LIN {X 0,Y 398.014,Z 934.007,A -85,B 0,C 180,E1 13512.725,E2 13512.725} C_VEL
LIN {X 0,Y 394.69,Z 940.929,A -85,B 0,C 180,E1 13512.435,E2 13512.435} C_VEL
LIN {X 0,Y 387.731,Z 954.302,A -85,B 0,C 180,E1 13511.831,E2 13511.831} C_VEL
LIN {X 0,Y 384.258,Z 960.422,A -85,B 0,C 180,E1 13511.522,E2 13511.522} C_VEL
LIN {X 0,Y 377.396,Z 971.989,A -85,B 0,C 180,E1 13510.92,E2 13510.92} C_VEL
LIN {X 0,Y 367.725,Z 986.837,A -85,B 0,C 180,E1 13510.022,E2 13510.022} C_VEL
LIN {X 0,Y 358.47,Z 999.7,A -85,B 0,C 180,E1 13509.091,E2 13509.091} C_VEL
LIN {X 0,Y 349.857,Z 1010.761,A -85,B 0,C 180,E1 13508.133,E2 13508.133} C_VEL
LIN {X 0,Y 342.33,Z 1019.858,A -85,B 0,C 180,E1 13507.215,E2 13507.215} C_VEL
LIN {X 0,Y 335.258,Z 1027.833,A -85,B 0,C 180,E1 13506.25,E2 13506.25} C_VEL
LIN {X 0,Y 328.859,Z 1034.776,A -85,B 0,C 180,E1 13505.234,E2 13505.234} C_VEL
LIN {X 0,Y 322.807,Z 1041.004,A -85,B 0,C 180,E1 13504.122,E2 13504.122} C_VEL
LIN {X 0,Y 317.742,Z 1046.055,A -85,B 0,C 180,E1 13503.067,E2 13503.067} C_VEL
LIN {X 0,Y 313.157,Z 1050.485,A -85,B 0,C 180,E1 13501.963,E2 13501.963} C_VEL
LIN {X 0,Y 312.58,Z 1051.188,A -85,B 0,C 180,E1 13501.741,E2 13501.741} C_VEL
LIN {X 0,Y 311.047,Z 1063.684,A -85,B 0,C 180,E1 13500.267,E2 13500.267} C_VEL
LIN {X 0,Y 309.538,Z 1073.557,A -85,B 0,C 180,E1 13498.797,E2 13498.797} C_VEL
LIN {X 0,Y 307.841,Z 1083.184,A -85,B 0,C 180,E1 13497.021,E2 13497.021} C_VEL
LIN {X 0,Y 306.001,Z 1091.827,A -85,B 0,C 180,E1 13494.938,E2 13494.938} C_VEL
LIN {X 0,Y 304.51,Z 1097.96,A -85,B 0,C 180,E1 13493.022,E2 13493.022} C_VEL
LIN {X 0,Y 303.205,Z 1102.729,A -85,B 0,C 180,E1 13491.084,E2 13491.084} C_VEL
LIN {X 0,Y 302.1,Z 1106.25,A -85,B 0,C 180,E1 13489.125,E2 13489.125} C_VEL
LIN {X 0,Y 301.125,Z 1108.835,A -85,B 0,C 180,E1 13486.95,E2 13486.95} C_VEL
LIN {X 0,Y 300.227,Z 1110.227,A -85,B 0,C 180,E1 13484.151,E2 13484.151} C_VEL
LIN {X 0,Y 299.753,Z 1109.674,A -85,B 0,C 180,E1 13481.726,E2 13481.726} C_VEL
LIN {X 0,Y 299.575,Z 1108.058,A -85,B 0,C 180,E1 13479.689,E2 13479.689} C_VEL
LIN {X 0,Y 299.582,Z 1105.256,A -85,B 0,C 180,E1 13477.6,E2 13477.6} C_VEL
LIN {X 0,Y 299.825,Z 1100.918,A -85,B 0,C 180,E1 13475.363,E2 13475.363} C_VEL
LIN {X 0,Y 300.406,Z 1093.744,A -85,B 0,C 180,E1 13472.714,E2 13472.714} C_VEL
LIN {X 0,Y 300.97,Z 1088.064,A -85,B 0,C 180,E1 13471.032,E2 13471.032} C_VEL
LIN {X 0,Y 302.662,Z 1088.577,A -85,B 0,C 180,E1 13470.076,E2 13470.076} C_VEL
LIN {X 0,Y 308.965,Z 1089.207,A -85,B 0,C 180,E1 13467.505,E2 13467.505} C_VEL
LIN {X 0,Y 318.43,Z 1089.392,A -85,B 0,C 180,E1 13464.485,E2 13464.485} C_VEL
LIN {X 0,Y 330.052,Z 1088.628,A -85,B 0,C 180,E1 13461.689,E2 13461.689} C_VEL
LIN {X 0,Y 343.834,Z 1086.815,A -85,B 0,C 180,E1 13459.132,E2 13459.132} C_VEL
LIN {X 0,Y 345.437,Z 1086.554,A -85,B 0,C 180,E1 13458.874,E2 13458.874} C_VEL
LIN {X 0,Y 335.157,Z 1103.247,A -85,B 0,C 180,E1 13455.24,E2 13455.24} C_VEL
LIN {X 0,Y 325.414,Z 1119.016,A -85,B 0,C 180,E1 13451.115,E2 13451.115} C_VEL
LIN {X 0,Y 317.973,Z 1131.208,A -85,B 0,C 180,E1 13447.29,E2 13447.29} C_VEL
LIN {X 0,Y 310.56,Z 1143.92,A -85,B 0,C 180,E1 13442.483,E2 13442.483} C_VEL
LIN {X 0,Y 305.641,Z 1152.997,A -85,B 0,C 180,E1 13438.32,E2 13438.32} C_VEL
LIN {X 0,Y 301.289,Z 1162.04,A -85,B 0,C 180,E1 13433.263,E2 13433.263} C_VEL
LIN {X 0,Y 298.782,Z 1168.154,A -85,B 0,C 180,E1 13428.944,E2 13428.944} C_VEL
LIN {X 0,Y 297.276,Z 1172.834,A -85,B 0,C 180,E1 13424.813,E2 13424.813} C_VEL
LIN {X 0,Y 296.351,Z 1176.957,A -85,B 0,C 180,E1 13419.865,E2 13419.865} C_VEL
LIN {X 0,Y 296.061,Z 1179.123,A -85,B 0,C 180,E1 13415.623,E2 13415.623} C_VEL
LIN {X 0,Y 295.995,Z 1180.069,A -85,B 0,C 180,E1 13411.938,E2 13411.938} C_VEL
LIN {X 0,Y 295.993,Z 1180.126,A -85,B 0,C 180,E1 13408.454,E2 13408.454} C_VEL
LIN {X 0,Y 296.038,Z 1179.362,A -85,B 0,C 180,E1 13404.964,E2 13404.964} C_VEL
LIN {X 0,Y 296.241,Z 1177.665,A -85,B 0,C 180,E1 13401.266,E2 13401.266} C_VEL
LIN {X 0,Y 296.743,Z 1174.897,A -85,B 0,C 180,E1 13397.351,E2 13397.351} C_VEL
LIN {X 0,Y 298.092,Z 1170.287,A -85,B 0,C 180,E1 13392.633,E2 13392.633} C_VEL
LIN {X 0,Y 300.451,Z 1163.965,A -85,B 0,C 180,E1 13387.913,E2 13387.913} C_VEL
LIN {X 0,Y 303.528,Z 1157.228,A -85,B 0,C 180,E1 13383.808,E2 13383.808} C_VEL
LIN {X 0,Y 308.813,Z 1147.142,A -85,B 0,C 180,E1 13378.801,E2 13378.801} C_VEL
LIN {X 0,Y 314.293,Z 1137.438,A -85,B 0,C 180,E1 13374.845,E2 13374.845} C_VEL
LIN {X 0,Y 321.668,Z 1125.291,A -85,B 0,C 180,E1 13370.649,E2 13370.649} C_VEL
LIN {X 0,Y 329.932,Z 1111.715,A -85,B 0,C 180,E1 13366.775,E2 13366.775} C_VEL
LIN {X 0,Y 339.348,Z 1096.62,A -85,B 0,C 180,E1 13363.125,E2 13363.125} C_VEL
LIN {X 0,Y 349.127,Z 1080.443,A -85,B 0,C 180,E1 13359.87,E2 13359.87} C_VEL
LIN {X 0,Y 359.711,Z 1062.568,A -85,B 0,C 180,E1 13356.821,E2 13356.821} C_VEL
LIN {X 0,Y 369.373,Z 1045.349,A -85,B 0,C 180,E1 13354.352,E2 13354.352} C_VEL
LIN {X 0,Y 372.803,Z 1039.126,A -85,B 0,C 180,E1 13353.53,E2 13353.53} C_VEL
LIN {X 0,Y 375.069,Z 1033.805,A -85,B 0,C 180,E1 13352.741,E2 13352.741} C_VEL
LIN {X 0,Y 378.793,Z 1021.008,A -85,B 0,C 180,E1 13350.448,E2 13350.448} C_VEL
LIN {X 0,Y 381.221,Z 1015.371,A -85,B 0,C 180,E1 13349.727,E2 13349.727} C_VEL
LIN {X 0,Y 391.468,Z 994.143,A -85,B 0,C 180,E1 13347.75,E2 13347.75} C_VEL
LIN {X 0,Y 401.494,Z 971.549,A -85,B 0,C 180,E1 13345.973,E2 13345.973} C_VEL
LIN {X 0,Y 410.028,Z 949.956,A -85,B 0,C 180,E1 13344.557,E2 13344.557} C_VEL
LIN {X 0,Y 418.764,Z 924.964,A -85,B 0,C 180,E1 13343.187,E2 13343.187} C_VEL
LIN {X 0,Y 425.429,Z 902.92,A -85,B 0,C 180,E1 13342.184,E2 13342.184} C_VEL
LIN {X 0,Y 432.132,Z 876.432,A -85,B 0,C 180,E1 13341.205,E2 13341.205} C_VEL
LIN {X 0,Y 440.836,Z 835.745,A -85,B 0,C 180,E1 13340.043,E2 13340.043} C_VEL
LIN {X 0,Y 454.676,Z 767.712,A -85,B 0,C 180,E1 13338.499,E2 13338.499} C_VEL
LIN {X 0,Y 466.705,Z 700.879,A -85,B 0,C 180,E1 13337.159,E2 13337.159} C_VEL
LIN {X 0,Y 476.357,Z 638.132,A -85,B 0,C 180,E1 13336.035,E2 13336.035} C_VEL
LIN {X 0,Y 480.624,Z 605.539,A -85,B 0,C 180,E1 13335.479,E2 13335.479} C_VEL
LIN {X 0,Y 475.05,Z 603.148,A -85,B 0,C 180,E1 13332.397,E2 13332.397} C_VEL
LIN {X 0,Y 471.241,Z 602.431,A -85,B 0,C 180,E1 13329.773,E2 13329.773} C_VEL
LIN {X 0,Y 467.289,Z 604.236,A -85,B 0,C 180,E1 13326.265,E2 13326.265} C_VEL
LIN {X 0,Y 465.287,Z 607.075,A -85,B 0,C 180,E1 13323.696,E2 13323.696} C_VEL
LIN {X 0,Y 463.897,Z 611.957,A -85,B 0,C 180,E1 13320.679,E2 13320.679} C_VEL
LIN {X 0,Y 463.503,Z 617.063,A -85,B 0,C 180,E1 13318.455,E2 13318.455} C_VEL
LIN {X 0,Y 460.723,Z 644.789,A -85,B 0,C 180,E1 13316.36,E2 13316.36} C_VEL
LIN {X 0,Y 457.571,Z 678.937,A -85,B 0,C 180,E1 13313.931,E2 13313.931} C_VEL
LIN {X 0,Y 455.045,Z 708.757,A -85,B 0,C 180,E1 13311.749,E2 13311.749} C_VEL
LIN {X 0,Y 453.418,Z 735.459,A -85,B 0,C 180,E1 13309.502,E2 13309.502} C_VEL
LIN {X 0,Y 452.74,Z 761.032,A -85,B 0,C 180,E1 13307.046,E2 13307.046} C_VEL
LIN {X 0,Y 453.158,Z 782.423,A -85,B 0,C 180,E1 13304.728,E2 13304.728} C_VEL
LIN {X 0,Y 454.662,Z 802.684,A -85,B 0,C 180,E1 13302.3,E2 13302.3} C_VEL
LIN {X 0,Y 455.41,Z 809.682,A -85,B 0,C 180,E1 13301.419,E2 13301.419} C_VEL
LIN {X 0,Y 445.885,Z 851.739,A -85,B 0,C 180,E1 13300.46,E2 13300.46} C_VEL
LIN {X 0,Y 436.683,Z 887.236,A -85,B 0,C 180,E1 13299.465,E2 13299.465} C_VEL
LIN {X 0,Y 426.541,Z 923.447,A -85,B 0,C 180,E1 13298.164,E2 13298.164} C_VEL
LIN {X 0,Y 416.365,Z 957.126,A -85,B 0,C 180,E1 13296.656,E2 13296.656} C_VEL
LIN {X 0,Y 408.565,Z 980.494,A -85,B 0,C 180,E1 13295.386,E2 13295.386} C_VEL
LIN {X 0,Y 400.463,Z 1001.95,A -85,B 0,C 180,E1 13294.003,E2 13294.003} C_VEL
LIN {X 0,Y 390.854,Z 1024.162,A -85,B 0,C 180,E1 13292.264,E2 13292.264} C_VEL
LIN {X 0,Y 380.916,Z 1044.801,A -85,B 0,C 180,E1 13290.321,E2 13290.321} C_VEL
LIN {X 0,Y 370.977,Z 1063.841,A -85,B 0,C 180,E1 13288.196,E2 13288.196} C_VEL
LIN {X 0,Y 360.474,Z 1082.231,A -85,B 0,C 180,E1 13285.73,E2 13285.73} C_VEL
LIN {X 0,Y 349.696,Z 1099.779,A -85,B 0,C 180,E1 13282.911,E2 13282.911} C_VEL
LIN {X 0,Y 339.669,Z 1115.345,A -85,B 0,C 180,E1 13279.935,E2 13279.935} C_VEL
LIN {X 0,Y 329.417,Z 1130.44,A -85,B 0,C 180,E1 13276.447,E2 13276.447} C_VEL
LIN {X 0,Y 320.032,Z 1143.814,A -85,B 0,C 180,E1 13272.682,E2 13272.682} C_VEL
LIN {X 0,Y 311.057,Z 1156.534,A -85,B 0,C 180,E1 13268.34,E2 13268.34} C_VEL
LIN {X 0,Y 303.649,Z 1167.257,A -85,B 0,C 180,E1 13263.811,E2 13263.811} C_VEL
LIN {X 0,Y 297.57,Z 1176.576,A -85,B 0,C 180,E1 13258.935,E2 13258.935} C_VEL
LIN {X 0,Y 293.003,Z 1184.34,A -85,B 0,C 180,E1 13253.743,E2 13253.743} C_VEL
LIN {X 0,Y 290.117,Z 1190.259,A -85,B 0,C 180,E1 13248.596,E2 13248.596} C_VEL
LIN {X 0,Y 288.587,Z 1194.684,A -85,B 0,C 180,E1 13243.42,E2 13243.42} C_VEL
LIN {X 0,Y 288.063,Z 1197.528,A -85,B 0,C 180,E1 13238.581,E2 13238.581} C_VEL
LIN {X 0,Y 287.98,Z 1198.959,A -85,B 0,C 180,E1 13234.179,E2 13234.179} C_VEL
LIN {X 0,Y 287.993,Z 1199.454,A -85,B 0,C 180,E1 13229.799,E2 13229.799} C_VEL
LIN {X 0,Y 287.98,Z 1198.913,A -85,B 0,C 180,E1 13225.617,E2 13225.617} C_VEL
LIN {X 0,Y 288.083,Z 1197.331,A -85,B 0,C 180,E1 13221.012,E2 13221.012} C_VEL
LIN {X 0,Y 288.668,Z 1194.394,A -85,B 0,C 180,E1 13216.17,E2 13216.17} C_VEL
LIN {X 0,Y 290.341,Z 1189.756,A -85,B 0,C 180,E1 13210.901,E2 13210.901} C_VEL
LIN {X 0,Y 293.445,Z 1183.493,A -85,B 0,C 180,E1 13205.649,E2 13205.649} C_VEL
LIN {X 0,Y 298.212,Z 1175.485,A -85,B 0,C 180,E1 13200.468,E2 13200.468} C_VEL
LIN {X 0,Y 304.495,Z 1166.011,A -85,B 0,C 180,E1 13195.609,E2 13195.609} C_VEL
LIN {X 0,Y 312.467,Z 1154.557,A -85,B 0,C 180,E1 13190.918,E2 13190.918} C_VEL
LIN {X 0,Y 321.663,Z 1141.485,A -85,B 0,C 180,E1 13186.606,E2 13186.606} C_VEL
LIN {X 0,Y 331.376,Z 1127.495,A -85,B 0,C 180,E1 13182.84,E2 13182.84} C_VEL
LIN {X 0,Y 342.245,Z 1111.347,A -85,B 0,C 180,E1 13179.264,E2 13179.264} C_VEL
LIN {X 0,Y 353.335,Z 1093.987,A -85,B 0,C 180,E1 13176.104,E2 13176.104} C_VEL
LIN {X 0,Y 364.079,Z 1075.99,A -85,B 0,C 180,E1 13173.393,E2 13173.393} C_VEL
LIN {X 0,Y 375.16,Z 1055.883,A -85,B 0,C 180,E1 13170.882,E2 13170.882} C_VEL
LIN {X 0,Y 385.523,Z 1035.367,A -85,B 0,C 180,E1 13168.759,E2 13168.759} C_VEL
LIN {X 0,Y 395.263,Z 1014.129,A -85,B 0,C 180,E1 13166.925,E2 13166.925} C_VEL
LIN {X 0,Y 404.293,Z 991.925,A -85,B 0,C 180,E1 13165.332,E2 13165.332} C_VEL
LIN {X 0,Y 412.504,Z 968.84,A -85,B 0,C 180,E1 13163.958,E2 13163.958} C_VEL
LIN {X 0,Y 422.561,Z 936.541,A -85,B 0,C 180,E1 13162.394,E2 13162.394} C_VEL
LIN {X 0,Y 432.734,Z 901.343,A -85,B 0,C 180,E1 13161.011,E2 13161.011} C_VEL
LIN {X 0,Y 442.358,Z 865.215,A -85,B 0,C 180,E1 13159.894,E2 13159.894} C_VEL
LIN {X 0,Y 448.761,Z 839.044,A -85,B 0,C 180,E1 13159.229,E2 13159.229} C_VEL
LIN {X 0,Y 440.38,Z 855.925,A -85,B 0,C 180,E1 13158.277,E2 13158.277} C_VEL
LIN {X 0,Y 436.828,Z 863.044,A -85,B 0,C 180,E1 13157.877,E2 13157.877} C_VEL
LIN {X 0,Y 428.321,Z 879.64,A -85,B 0,C 180,E1 13156.903,E2 13156.903} C_VEL
LIN {X 0,Y 424.296,Z 887.378,A -85,B 0,C 180,E1 13156.434,E2 13156.434} C_VEL
LIN {X 0,Y 416.15,Z 902.746,A -85,B 0,C 180,E1 13155.468,E2 13155.468} C_VEL
LIN {X 0,Y 405.614,Z 923.215,A -85,B 0,C 180,E1 13154.348,E2 13154.348} C_VEL
LIN {X 0,Y 398.353,Z 937.989,A -85,B 0,C 180,E1 13153.734,E2 13153.734} C_VEL
LIN {X 0,Y 389.653,Z 954.885,A -85,B 0,C 180,E1 13153.051,E2 13153.051} C_VEL
LIN {X 0,Y 384.55,Z 963.752,A -85,B 0,C 180,E1 13152.616,E2 13152.616} C_VEL
LIN {X 0,Y 377.206,Z 975.718,A -85,B 0,C 180,E1 13151.998,E2 13151.998} C_VEL
LIN {X 0,Y 367.979,Z 989.516,A -85,B 0,C 180,E1 13151.203,E2 13151.203} C_VEL
LIN {X 0,Y 358.299,Z 1002.633,A -85,B 0,C 180,E1 13150.288,E2 13150.288} C_VEL
LIN {X 0,Y 349.026,Z 1014.167,A -85,B 0,C 180,E1 13149.315,E2 13149.315} C_VEL
LIN {X 0,Y 341.264,Z 1023.234,A -85,B 0,C 180,E1 13148.424,E2 13148.424} C_VEL
LIN {X 0,Y 333.496,Z 1031.746,A -85,B 0,C 180,E1 13147.407,E2 13147.407} C_VEL
LIN {X 0,Y 326.372,Z 1039.06,A -85,B 0,C 180,E1 13146.332,E2 13146.332} C_VEL
LIN {X 0,Y 320.329,Z 1045.099,A -85,B 0,C 180,E1 13145.276,E2 13145.276} C_VEL
LIN {X 0,Y 314.812,Z 1050.293,A -85,B 0,C 180,E1 13144.184,E2 13144.184} C_VEL
LIN {X 0,Y 309.371,Z 1055.333,A -85,B 0,C 180,E1 13142.907,E2 13142.907} C_VEL
LIN {X 0,Y 305.378,Z 1058.923,A -85,B 0,C 180,E1 13141.876,E2 13141.876} C_VEL
LIN {X 0,Y 304.821,Z 1059.658,A -85,B 0,C 180,E1 13141.645,E2 13141.645} C_VEL
LIN {X 0,Y 302.974,Z 1071.89,A -85,B 0,C 180,E1 13139.945,E2 13139.945} C_VEL
LIN {X 0,Y 301.247,Z 1081.202,A -85,B 0,C 180,E1 13138.288,E2 13138.288} C_VEL
LIN {X 0,Y 299.578,Z 1089.042,A -85,B 0,C 180,E1 13136.556,E2 13136.556} C_VEL
LIN {X 0,Y 297.743,Z 1096.741,A -85,B 0,C 180,E1 13134.411,E2 13134.411} C_VEL
LIN {X 0,Y 295.893,Z 1103.131,A -85,B 0,C 180,E1 13131.947,E2 13131.947} C_VEL
LIN {X 0,Y 294.592,Z 1107.034,A -85,B 0,C 180,E1 13129.834,E2 13129.834} C_VEL
LIN {X 0,Y 293.583,Z 1109.561,A -85,B 0,C 180,E1 13127.81,E2 13127.81} C_VEL
LIN {X 0,Y 292.779,Z 1110.991,A -85,B 0,C 180,E1 13125.765,E2 13125.765} C_VEL
LIN {X 0,Y 292.193,Z 1111.364,A -85,B 0,C 180,E1 13123.704,E2 13123.704} C_VEL
LIN {X 0,Y 291.808,Z 1110.667,A -85,B 0,C 180,E1 13121.625,E2 13121.625} C_VEL
LIN {X 0,Y 291.624,Z 1108.651,A -85,B 0,C 180,E1 13119.319,E2 13119.319} C_VEL
LIN {X 0,Y 291.718,Z 1104.507,A -85,B 0,C 180,E1 13116.572,E2 13116.572} C_VEL
LIN {X 0,Y 292.073,Z 1099.16,A -85,B 0,C 180,E1 13114.209,E2 13114.209} C_VEL
LIN {X 0,Y 292.669,Z 1092.631,A -85,B 0,C 180,E1 13111.958,E2 13111.958} C_VEL
LIN {X 0,Y 294.265,Z 1093.219,A -85,B 0,C 180,E1 13110.928,E2 13110.928} C_VEL
LIN {X 0,Y 300.147,Z 1094.066,A -85,B 0,C 180,E1 13108.241,E2 13108.241} C_VEL
LIN {X 0,Y 309.579,Z 1094.484,A -85,B 0,C 180,E1 13104.906,E2 13104.906} C_VEL
LIN {X 0,Y 320.998,Z 1093.948,A -85,B 0,C 180,E1 13101.92,E2 13101.92} C_VEL
LIN {X 0,Y 334.828,Z 1092.438,A -85,B 0,C 180,E1 13099.156,E2 13099.156} C_VEL
LIN {X 0,Y 336.547,Z 1092.354,A -85,B 0,C 180,E1 13098.802,E2 13098.802} C_VEL
LIN {X 0,Y 326.253,Z 1108.519,A -85,B 0,C 180,E1 13095.071,E2 13095.071} C_VEL
LIN {X 0,Y 316.861,Z 1122.956,A -85,B 0,C 180,E1 13091.026,E2 13091.026} C_VEL
LIN {X 0,Y 308.275,Z 1136.549,A -85,B 0,C 180,E1 13086.412,E2 13086.412} C_VEL
LIN {X 0,Y 302.07,Z 1146.789,A -85,B 0,C 180,E1 13082.206,E2 13082.206} C_VEL
LIN {X 0,Y 296.312,Z 1157.145,A -85,B 0,C 180,E1 13077.018,E2 13077.018} C_VEL
LIN {X 0,Y 292.881,Z 1164.103,A -85,B 0,C 180,E1 13072.694,E2 13072.694} C_VEL
LIN {X 0,Y 290.325,Z 1170.426,A -85,B 0,C 180,E1 13067.852,E2 13067.852} C_VEL
LIN {X 0,Y 288.843,Z 1175.088,A -85,B 0,C 180,E1 13063.006,E2 13063.006} C_VEL
LIN {X 0,Y 288.275,Z 1177.873,A -85,B 0,C 180,E1 13058.982,E2 13058.982} C_VEL
LIN {X 0,Y 288.051,Z 1179.591,A -85,B 0,C 180,E1 13055.18,E2 13055.18} C_VEL
LIN {X 0,Y 287.997,Z 1180.377,A -85,B 0,C 180,E1 13051.594,E2 13051.594} C_VEL
LIN {X 0,Y 288,Z 1180.344,A -85,B 0,C 180,E1 13048.013,E2 13048.013} C_VEL
LIN {X 0,Y 288.061,Z 1179.491,A -85,B 0,C 180,E1 13044.425,E2 13044.425} C_VEL
LIN {X 0,Y 288.304,Z 1177.709,A -85,B 0,C 180,E1 13040.621,E2 13040.621} C_VEL
LIN {X 0,Y 289.106,Z 1174.226,A -85,B 0,C 180,E1 13035.788,E2 13035.788} C_VEL
LIN {X 0,Y 290.795,Z 1169.062,A -85,B 0,C 180,E1 13030.937,E2 13030.937} C_VEL
LIN {X 0,Y 293.23,Z 1163.369,A -85,B 0,C 180,E1 13026.703,E2 13026.703} C_VEL
LIN {X 0,Y 297.462,Z 1155.059,A -85,B 0,C 180,E1 13021.712,E2 13021.712} C_VEL
LIN {X 0,Y 302.72,Z 1145.684,A -85,B 0,C 180,E1 13017.204,E2 13017.204} C_VEL
LIN {X 0,Y 309.427,Z 1134.853,A -85,B 0,C 180,E1 13012.827,E2 13012.827} C_VEL
LIN {X 0,Y 317.472,Z 1122.037,A -85,B 0,C 180,E1 13008.597,E2 13008.597} C_VEL
LIN {X 0,Y 326.533,Z 1108.194,A -85,B 0,C 180,E1 13004.735,E2 13004.735} C_VEL
LIN {X 0,Y 336.251,Z 1092.902,A -85,B 0,C 180,E1 13001.212,E2 13001.212} C_VEL
LIN {X 0,Y 346.526,Z 1076.682,A -85,B 0,C 180,E1 12998.03,E2 12998.03} C_VEL
LIN {X 0,Y 357.37,Z 1058.563,A -85,B 0,C 180,E1 12995.081,E2 12995.081} C_VEL
LIN {X 0,Y 368.737,Z 1038.738,A -85,B 0,C 180,E1 12992.367,E2 12992.367} C_VEL
LIN {X 0,Y 378.852,Z 1019.807,A -85,B 0,C 180,E1 12990.196,E2 12990.196} C_VEL
LIN {X 0,Y 381.221,Z 1015.371,A -85,B 0,C 180,E1 12989.727,E2 12989.727} C_VEL
LIN {X 0,Y 383.63,Z 1009.691,A -85,B 0,C 180,E1 12989.025,E2 12989.025} C_VEL
LIN {X 0,Y 387.595,Z 995.885,A -85,B 0,C 180,E1 12986.93,E2 12986.93} C_VEL
LIN {X 0,Y 390.035,Z 989.923,A -85,B 0,C 180,E1 12986.29,E2 12986.29} C_VEL
LIN {X 0,Y 399.447,Z 968.502,A -85,B 0,C 180,E1 12984.686,E2 12984.686} C_VEL
LIN {X 0,Y 408.62,Z 945.55,A -85,B 0,C 180,E1 12983.231,E2 12983.231} C_VEL
LIN {X 0,Y 416.974,Z 921.32,A -85,B 0,C 180,E1 12981.968,E2 12981.968} C_VEL
LIN {X 0,Y 424.734,Z 894.931,A -85,B 0,C 180,E1 12980.844,E2 12980.844} C_VEL
LIN {X 0,Y 431.12,Z 868.513,A -85,B 0,C 180,E1 12979.947,E2 12979.947} C_VEL
LIN {X 0,Y 440.685,Z 824.326,A -85,B 0,C 180,E1 12978.776,E2 12978.776} C_VEL
LIN {X 0,Y 454.489,Z 756.835,A -85,B 0,C 180,E1 12977.298,E2 12977.298} C_VEL
LIN {X 0,Y 466.083,Z 692.135,A -85,B 0,C 180,E1 12976.043,E2 12976.043} C_VEL
LIN {X 0,Y 475.398,Z 630.7,A -85,B 0,C 180,E1 12974.973,E2 12974.973} C_VEL
LIN {X 0,Y 477.78,Z 612.645,A -85,B 0,C 180,E1 12974.669,E2 12974.669} C_VEL
LIN {X 0,Y 471.735,Z 610.463,A -85,B 0,C 180,E1 12970.997,E2 12970.997} C_VEL
LIN {X 0,Y 469.775,Z 610.503,A -85,B 0,C 180,E1 12969.556,E2 12969.556} C_VEL
LIN {X 0,Y 466.175,Z 612.244,A -85,B 0,C 180,E1 12966.28,E2 12966.28} C_VEL
LIN {X 0,Y 464.276,Z 614.951,A -85,B 0,C 180,E1 12963.828,E2 12963.828} C_VEL
LIN {X 0,Y 462.901,Z 619.763,A -85,B 0,C 180,E1 12960.866,E2 12960.866} C_VEL
LIN {X 0,Y 462.481,Z 623.861,A -85,B 0,C 180,E1 12959.086,E2 12959.086} C_VEL
LIN {X 0,Y 458.864,Z 656.466,A -85,B 0,C 180,E1 12956.651,E2 12956.651} C_VEL
LIN {X 0,Y 453.696,Z 707.234,A -85,B 0,C 180,E1 12953.014,E2 12953.014} C_VEL
LIN {X 0,Y 451.594,Z 733.311,A -85,B 0,C 180,E1 12950.874,E2 12950.874} C_VEL
LIN {X 0,Y 450.341,Z 757.303,A -85,B 0,C 180,E1 12948.652,E2 12948.652} C_VEL
LIN {X 0,Y 450.094,Z 783.869,A -85,B 0,C 180,E1 12945.839,E2 12945.839} C_VEL
LIN {X 0,Y 451.246,Z 806.631,A -85,B 0,C 180,E1 12943.109,E2 12943.109} C_VEL
LIN {X 0,Y 451.841,Z 813.134,A -85,B 0,C 180,E1 12942.293,E2 12942.293} C_VEL
LIN {X 0,Y 442.11,Z 854.607,A -85,B 0,C 180,E1 12941.348,E2 12941.348} C_VEL
LIN {X 0,Y 432.258,Z 891.855,A -85,B 0,C 180,E1 12940.292,E2 12940.292} C_VEL
LIN {X 0,Y 422.263,Z 926.666,A -85,B 0,C 180,E1 12939.028,E2 12939.028} C_VEL
LIN {X 0,Y 411.783,Z 960.528,A -85,B 0,C 180,E1 12937.501,E2 12937.501} C_VEL
LIN {X 0,Y 403.733,Z 983.613,A -85,B 0,C 180,E1 12936.221,E2 12936.221} C_VEL
LIN {X 0,Y 395.071,Z 1005.133,A -85,B 0,C 180,E1 12934.79,E2 12934.79} C_VEL
LIN {X 0,Y 386.015,Z 1025.532,A -85,B 0,C 180,E1 12933.181,E2 12933.181} C_VEL
LIN {X 0,Y 375.478,Z 1046.604,A -85,B 0,C 180,E1 12931.172,E2 12931.172} C_VEL
LIN {X 0,Y 364.771,Z 1066.143,A -85,B 0,C 180,E1 12928.933,E2 12928.933} C_VEL
LIN {X 0,Y 353.987,Z 1084.438,A -85,B 0,C 180,E1 12926.431,E2 12926.431} C_VEL
LIN {X 0,Y 342.948,Z 1101.76,A -85,B 0,C 180,E1 12923.576,E2 12923.576} C_VEL
LIN {X 0,Y 332.169,Z 1117.662,A -85,B 0,C 180,E1 12920.404,E2 12920.404} C_VEL
LIN {X 0,Y 321.805,Z 1132.381,A -85,B 0,C 180,E1 12916.877,E2 12916.877} C_VEL
LIN {X 0,Y 312.194,Z 1145.64,A -85,B 0,C 180,E1 12913.011,E2 12913.011} C_VEL
LIN {X 0,Y 303.41,Z 1157.484,A -85,B 0,C 180,E1 12908.763,E2 12908.763} C_VEL
LIN {X 0,Y 295.54,Z 1168.424,A -85,B 0,C 180,E1 12903.931,E2 12903.931} C_VEL
LIN {X 0,Y 289.191,Z 1177.765,A -85,B 0,C 180,E1 12898.721,E2 12898.721} C_VEL
LIN {X 0,Y 284.823,Z 1185.039,A -85,B 0,C 180,E1 12893.588,E2 12893.588} C_VEL
LIN {X 0,Y 281.889,Z 1191,A -85,B 0,C 180,E1 12888.079,E2 12888.079} C_VEL
LIN {X 0,Y 280.506,Z 1194.951,A -85,B 0,C 180,E1 12882.975,E2 12882.975} C_VEL
LIN {X 0,Y 280.042,Z 1197.561,A -85,B 0,C 180,E1 12878.002,E2 12878.002} C_VEL
LIN {X 0,Y 279.986,Z 1198.831,A -85,B 0,C 180,E1 12873.683,E2 12873.683} C_VEL
LIN {X 0,Y 279.995,Z 1199.152,A -85,B 0,C 180,E1 12869.25,E2 12869.25} C_VEL
LIN {X 0,Y 279.984,Z 1198.554,A -85,B 0,C 180,E1 12865.081,E2 12865.081} C_VEL
LIN {X 0,Y 280.126,Z 1196.84,A -85,B 0,C 180,E1 12860.34,E2 12860.34} C_VEL
LIN {X 0,Y 280.898,Z 1193.667,A -85,B 0,C 180,E1 12855.147,E2 12855.147} C_VEL
LIN {X 0,Y 282.855,Z 1188.794,A -85,B 0,C 180,E1 12849.729,E2 12849.729} C_VEL
LIN {X 0,Y 286.372,Z 1182.299,A -85,B 0,C 180,E1 12844.342,E2 12844.342} C_VEL
LIN {X 0,Y 291.759,Z 1173.87,A -85,B 0,C 180,E1 12838.957,E2 12838.957} C_VEL
LIN {X 0,Y 298.789,Z 1163.828,A -85,B 0,C 180,E1 12833.913,E2 12833.913} C_VEL
LIN {X 0,Y 307.088,Z 1152.503,A -85,B 0,C 180,E1 12829.346,E2 12829.346} C_VEL
LIN {X 0,Y 316.865,Z 1139.176,A -85,B 0,C 180,E1 12825.019,E2 12825.019} C_VEL
LIN {X 0,Y 327.146,Z 1124.861,A -85,B 0,C 180,E1 12821.245,E2 12821.245} C_VEL
LIN {X 0,Y 338.549,Z 1108.283,A -85,B 0,C 180,E1 12817.669,E2 12817.669} C_VEL
LIN {X 0,Y 350.097,Z 1090.523,A -85,B 0,C 180,E1 12814.527,E2 12814.527} C_VEL
LIN {X 0,Y 361.324,Z 1072.084,A -85,B 0,C 180,E1 12811.834,E2 12811.834} C_VEL
LIN {X 0,Y 372.495,Z 1052.072,A -85,B 0,C 180,E1 12809.421,E2 12809.421} C_VEL
LIN {X 0,Y 383.121,Z 1031.276,A -85,B 0,C 180,E1 12807.344,E2 12807.344} C_VEL
LIN {X 0,Y 393.316,Z 1009.128,A -85,B 0,C 180,E1 12805.511,E2 12805.511} C_VEL
LIN {X 0,Y 402.639,Z 986.298,A -85,B 0,C 180,E1 12803.952,E2 12803.952} C_VEL
LIN {X 0,Y 410.669,Z 963.496,A -85,B 0,C 180,E1 12802.661,E2 12802.661} C_VEL
LIN {X 0,Y 421.216,Z 929.649,A -85,B 0,C 180,E1 12801.105,E2 12801.105} C_VEL
LIN {X 0,Y 431.257,Z 895.039,A -85,B 0,C 180,E1 12799.82,E2 12799.82} C_VEL
LIN {X 0,Y 439.459,Z 864.388,A -85,B 0,C 180,E1 12798.899,E2 12798.899} C_VEL
LIN {X 0,Y 430.817,Z 881.146,A -85,B 0,C 180,E1 12797.98,E2 12797.98} C_VEL
LIN {X 0,Y 425.874,Z 890.299,A -85,B 0,C 180,E1 12797.419,E2 12797.419} C_VEL
LIN {X 0,Y 417.508,Z 905.742,A -85,B 0,C 180,E1 12796.487,E2 12796.487} C_VEL
LIN {X 0,Y 414.318,Z 911.672,A -85,B 0,C 180,E1 12796.153,E2 12796.153} C_VEL
LIN {X 0,Y 406.83,Z 926.023,A -85,B 0,C 180,E1 12795.393,E2 12795.393} C_VEL
LIN {X 0,Y 399.167,Z 941.236,A -85,B 0,C 180,E1 12794.778,E2 12794.778} C_VEL
LIN {X 0,Y 390.874,Z 956.968,A -85,B 0,C 180,E1 12794.18,E2 12794.18} C_VEL
LIN {X 0,Y 385.501,Z 966.155,A -85,B 0,C 180,E1 12793.743,E2 12793.743} C_VEL
LIN {X 0,Y 377.869,Z 978.346,A -85,B 0,C 180,E1 12793.147,E2 12793.147} C_VEL
LIN {X 0,Y 367.971,Z 992.762,A -85,B 0,C 180,E1 12792.342,E2 12792.342} C_VEL
LIN {X 0,Y 357.874,Z 1006.076,A -85,B 0,C 180,E1 12791.442,E2 12791.442} C_VEL
LIN {X 0,Y 348.348,Z 1017.567,A -85,B 0,C 180,E1 12790.502,E2 12790.502} C_VEL
LIN {X 0,Y 340.342,Z 1026.586,A -85,B 0,C 180,E1 12789.64,E2 12789.64} C_VEL
LIN {X 0,Y 332.311,Z 1035.119,A -85,B 0,C 180,E1 12788.653,E2 12788.653} C_VEL
LIN {X 0,Y 324.816,Z 1042.561,A -85,B 0,C 180,E1 12787.588,E2 12787.588} C_VEL
LIN {X 0,Y 317.319,Z 1049.618,A -85,B 0,C 180,E1 12786.332,E2 12786.332} C_VEL
LIN {X 0,Y 311.227,Z 1055.183,A -85,B 0,C 180,E1 12785.144,E2 12785.144} C_VEL
LIN {X 0,Y 305.795,Z 1059.905,A -85,B 0,C 180,E1 12783.937,E2 12783.937} C_VEL
LIN {X 0,Y 301.337,Z 1063.737,A -85,B 0,C 180,E1 12782.812,E2 12782.812} C_VEL
LIN {X 0,Y 298.013,Z 1066.561,A -85,B 0,C 180,E1 12781.923,E2 12781.923} C_VEL
LIN {X 0,Y 296.945,Z 1067.648,A -85,B 0,C 180,E1 12781.495,E2 12781.495} C_VEL
LIN {X 0,Y 295.165,Z 1077.599,A -85,B 0,C 180,E1 12779.903,E2 12779.903} C_VEL
LIN {X 0,Y 293.005,Z 1087.662,A -85,B 0,C 180,E1 12777.849,E2 12777.849} C_VEL
LIN {X 0,Y 291.11,Z 1095.149,A -85,B 0,C 180,E1 12775.864,E2 12775.864} C_VEL
LIN {X 0,Y 289.55,Z 1100.635,A -85,B 0,C 180,E1 12774.024,E2 12774.024} C_VEL
LIN {X 0,Y 288.061,Z 1105.265,A -85,B 0,C 180,E1 12772.019,E2 12772.019} C_VEL
LIN {X 0,Y 286.772,Z 1108.747,A -85,B 0,C 180,E1 12769.96,E2 12769.96} C_VEL
LIN {X 0,Y 285.605,Z 1111.304,A -85,B 0,C 180,E1 12767.632,E2 12767.632} C_VEL
LIN {X 0,Y 284.542,Z 1112.609,A -85,B 0,C 180,E1 12764.719,E2 12764.719} C_VEL
LIN {X 0,Y 283.957,Z 1112.01,A -85,B 0,C 180,E1 12762.16,E2 12762.16} C_VEL
LIN {X 0,Y 283.711,Z 1110.36,A -85,B 0,C 180,E1 12760.01,E2 12760.01} C_VEL
LIN {X 0,Y 283.676,Z 1107.585,A -85,B 0,C 180,E1 12757.843,E2 12757.843} C_VEL
LIN {X 0,Y 283.895,Z 1103.157,A -85,B 0,C 180,E1 12755.443,E2 12755.443} C_VEL
LIN {X 0,Y 284.423,Z 1097.12,A -85,B 0,C 180,E1 12752.955,E2 12752.955} C_VEL
LIN {X 0,Y 286.045,Z 1097.691,A -85,B 0,C 180,E1 12751.842,E2 12751.842} C_VEL
LIN {X 0,Y 293.802,Z 1098.92,A -85,B 0,C 180,E1 12747.933,E2 12747.933} C_VEL
LIN {X 0,Y 304.956,Z 1099.359,A -85,B 0,C 180,E1 12744.062,E2 12744.062} C_VEL
LIN {X 0,Y 317.3,Z 1098.764,A -85,B 0,C 180,E1 12740.931,E2 12740.931} C_VEL
LIN {X 0,Y 327.86,Z 1097.768,A -85,B 0,C 180,E1 12738.795,E2 12738.795} C_VEL
LIN {X 0,Y 317.717,Z 1112.781,A -85,B 0,C 180,E1 12735.083,E2 12735.083} C_VEL
LIN {X 0,Y 308.296,Z 1126.876,A -85,B 0,C 180,E1 12730.914,E2 12730.914} C_VEL
LIN {X 0,Y 299.993,Z 1139.324,A -85,B 0,C 180,E1 12726.392,E2 12726.392} C_VEL
LIN {X 0,Y 293.279,Z 1150.12,A -85,B 0,C 180,E1 12721.673,E2 12721.673} C_VEL
LIN {X 0,Y 288.071,Z 1159.03,A -85,B 0,C 180,E1 12716.825,E2 12716.825} C_VEL
LIN {X 0,Y 284.308,Z 1166.565,A -85,B 0,C 180,E1 12711.802,E2 12711.802} C_VEL
LIN {X 0,Y 281.878,Z 1172.38,A -85,B 0,C 180,E1 12706.7,E2 12706.7} C_VEL
LIN {X 0,Y 280.758,Z 1175.993,A -85,B 0,C 180,E1 12702.55,E2 12702.55} C_VEL
LIN {X 0,Y 280.234,Z 1178.592,A -85,B 0,C 180,E1 12698.414,E2 12698.414} C_VEL
LIN {X 0,Y 280.027,Z 1180.395,A -85,B 0,C 180,E1 12693.688,E2 12693.688} C_VEL
LIN {X 0,Y 279.996,Z 1180.743,A -85,B 0,C 180,E1 12689.184,E2 12689.184} C_VEL
LIN {X 0,Y 280.047,Z 1180.025,A -85,B 0,C 180,E1 12685.087,E2 12685.087} C_VEL
LIN {X 0,Y 280.265,Z 1178.422,A -85,B 0,C 180,E1 12681.178,E2 12681.178} C_VEL
LIN {X 0,Y 280.781,Z 1175.91,A -85,B 0,C 180,E1 12677.247,E2 12677.247} C_VEL
LIN {X 0,Y 281.917,Z 1172.28,A -85,B 0,C 180,E1 12673.095,E2 12673.095} C_VEL
LIN {X 0,Y 284.436,Z 1166.306,A -85,B 0,C 180,E1 12667.908,E2 12667.908} C_VEL
LIN {X 0,Y 288.005,Z 1159.161,A -85,B 0,C 180,E1 12663.158,E2 12663.158} C_VEL
LIN {X 0,Y 292.801,Z 1150.902,A -85,B 0,C 180,E1 12658.62,E2 12658.62} C_VEL
LIN {X 0,Y 299.557,Z 1140.049,A -85,B 0,C 180,E1 12653.789,E2 12653.789} C_VEL
LIN {X 0,Y 306.694,Z 1129.267,A -85,B 0,C 180,E1 12649.799,E2 12649.799} C_VEL
LIN {X 0,Y 316.253,Z 1115.037,A -85,B 0,C 180,E1 12645.425,E2 12645.425} C_VEL
LIN {X 0,Y 325.883,Z 1100.796,A -85,B 0,C 180,E1 12641.795,E2 12641.795} C_VEL
LIN {X 0,Y 336.581,Z 1084.562,A -85,B 0,C 180,E1 12638.351,E2 12638.351} C_VEL
LIN {X 0,Y 346.563,Z 1068.957,A -85,B 0,C 180,E1 12635.554,E2 12635.554} C_VEL
LIN {X 0,Y 357.869,Z 1050.397,A -85,B 0,C 180,E1 12632.759,E2 12632.759} C_VEL
LIN {X 0,Y 367.301,Z 1034.041,A -85,B 0,C 180,E1 12630.662,E2 12630.662} C_VEL
LIN {X 0,Y 379.171,Z 1011.913,A -85,B 0,C 180,E1 12628.27,E2 12628.27} C_VEL
LIN {X 0,Y 388.795,Z 992.43,A -85,B 0,C 180,E1 12626.501,E2 12626.501} C_VEL
LIN {X 0,Y 390.035,Z 989.923,A -85,B 0,C 180,E1 12626.29,E2 12626.29} C_VEL
LIN {X 0,Y 392.491,Z 983.908,A -85,B 0,C 180,E1 12625.667,E2 12625.667} C_VEL
LIN {X 0,Y 396.587,Z 969.193,A -85,B 0,C 180,E1 12623.766,E2 12623.766} C_VEL
LIN {X 0,Y 398.812,Z 962.847,A -85,B 0,C 180,E1 12623.211,E2 12623.211} C_VEL
LIN {X 0,Y 408.102,Z 938.86,A -85,B 0,C 180,E1 12621.791,E2 12621.791} C_VEL
LIN {X 0,Y 416.519,Z 913.858,A -85,B 0,C 180,E1 12620.58,E2 12620.58} C_VEL
LIN {X 0,Y 423.496,Z 889.406,A -85,B 0,C 180,E1 12619.608,E2 12619.608} C_VEL
LIN {X 0,Y 430.89,Z 857.605,A -85,B 0,C 180,E1 12618.617,E2 12618.617} C_VEL
LIN {X 0,Y 442.203,Z 806.427,A -85,B 0,C 180,E1 12617.374,E2 12617.374} C_VEL
LIN {X 0,Y 455.207,Z 742.035,A -85,B 0,C 180,E1 12616.021,E2 12616.021} C_VEL
LIN {X 0,Y 466.31,Z 678.954,A -85,B 0,C 180,E1 12614.846,E2 12614.846} C_VEL
LIN {X 0,Y 474.996,Z 619.88,A -85,B 0,C 180,E1 12613.843,E2 12613.843} C_VEL
LIN {X 0,Y 469.419,Z 618.203,A -85,B 0,C 180,E1 12610.183,E2 12610.183} C_VEL
LIN {X 0,Y 465.161,Z 620.101,A -85,B 0,C 180,E1 12606.418,E2 12606.418} C_VEL
LIN {X 0,Y 463.231,Z 622.821,A -85,B 0,C 180,E1 12603.961,E2 12603.961} C_VEL
LIN {X 0,Y 461.827,Z 627.557,A -85,B 0,C 180,E1 12601.054,E2 12601.054} C_VEL
LIN {X 0,Y 461.448,Z 630.692,A -85,B 0,C 180,E1 12599.721,E2 12599.721} C_VEL
LIN {X 0,Y 457.437,Z 663.325,A -85,B 0,C 180,E1 12597.303,E2 12597.303} C_VEL
LIN {X 0,Y 452.054,Z 710.789,A -85,B 0,C 180,E1 12593.897,E2 12593.897} C_VEL
LIN {X 0,Y 449.564,Z 737.493,A -85,B 0,C 180,E1 12591.702,E2 12591.702} C_VEL
LIN {X 0,Y 447.88,Z 762.647,A -85,B 0,C 180,E1 12589.354,E2 12589.354} C_VEL
LIN {X 0,Y 447.245,Z 789.077,A -85,B 0,C 180,E1 12586.525,E2 12586.525} C_VEL
LIN {X 0,Y 448.069,Z 812.08,A -85,B 0,C 180,E1 12583.736,E2 12583.736} C_VEL
LIN {X 0,Y 448.335,Z 816.53,A -85,B 0,C 180,E1 12583.179,E2 12583.179} C_VEL
LIN {X 0,Y 437.715,Z 860.499,A -85,B 0,C 180,E1 12582.175,E2 12582.175} C_VEL
LIN {X 0,Y 427.717,Z 897.087,A -85,B 0,C 180,E1 12581.112,E2 12581.112} C_VEL
LIN {X 0,Y 417.132,Z 932.794,A -85,B 0,C 180,E1 12579.785,E2 12579.785} C_VEL
LIN {X 0,Y 407.503,Z 962.929,A -85,B 0,C 180,E1 12578.404,E2 12578.404} C_VEL
LIN {X 0,Y 399.61,Z 984.962,A -85,B 0,C 180,E1 12577.18,E2 12577.18} C_VEL
LIN {X 0,Y 390.494,Z 1006.844,A -85,B 0,C 180,E1 12575.716,E2 12575.716} C_VEL
LIN {X 0,Y 380.275,Z 1028.649,A -85,B 0,C 180,E1 12573.953,E2 12573.953} C_VEL
LIN {X 0,Y 370.124,Z 1048.398,A -85,B 0,C 180,E1 12572.048,E2 12572.048} C_VEL
LIN {X 0,Y 359.175,Z 1067.631,A -85,B 0,C 180,E1 12569.807,E2 12569.807} C_VEL
LIN {X 0,Y 347.816,Z 1086.064,A -85,B 0,C 180,E1 12567.227,E2 12567.227} C_VEL
LIN {X 0,Y 336.78,Z 1102.879,A -85,B 0,C 180,E1 12564.414,E2 12564.414} C_VEL
LIN {X 0,Y 325.756,Z 1118.583,A -85,B 0,C 180,E1 12561.223,E2 12561.223} C_VEL
LIN {X 0,Y 315.127,Z 1133.003,A -85,B 0,C 180,E1 12557.668,E2 12557.668} C_VEL
LIN {X 0,Y 305.621,Z 1145.679,A -85,B 0,C 180,E1 12553.911,E2 12553.911} C_VEL
LIN {X 0,Y 296.142,Z 1158.014,A -85,B 0,C 180,E1 12549.398,E2 12549.398} C_VEL
LIN {X 0,Y 288.301,Z 1168.379,A -85,B 0,C 180,E1 12544.662,E2 12544.662} C_VEL
LIN {X 0,Y 281.659,Z 1177.717,A -85,B 0,C 180,E1 12539.331,E2 12539.331} C_VEL
LIN {X 0,Y 276.927,Z 1185.174,A -85,B 0,C 180,E1 12533.85,E2 12533.85} C_VEL
LIN {X 0,Y 273.987,Z 1190.857,A -85,B 0,C 180,E1 12528.405,E2 12528.405} C_VEL
LIN {X 0,Y 272.529,Z 1194.809,A -85,B 0,C 180,E1 12523.146,E2 12523.146} C_VEL
LIN {X 0,Y 272.045,Z 1197.363,A -85,B 0,C 180,E1 12518.026,E2 12518.026} C_VEL
LIN {X 0,Y 271.991,Z 1198.66,A -85,B 0,C 180,E1 12513.369,E2 12513.369} C_VEL
LIN {X 0,Y 272.003,Z 1198.87,A -85,B 0,C 180,E1 12508.944,E2 12508.944} C_VEL
LIN {X 0,Y 271.991,Z 1198.192,A -85,B 0,C 180,E1 12504.513,E2 12504.513} C_VEL
LIN {X 0,Y 272.181,Z 1196.345,A -85,B 0,C 180,E1 12499.627,E2 12499.627} C_VEL
LIN {X 0,Y 273.111,Z 1193.053,A -85,B 0,C 180,E1 12494.278,E2 12494.278} C_VEL
LIN {X 0,Y 275.344,Z 1188.045,A -85,B 0,C 180,E1 12488.704,E2 12488.704} C_VEL
LIN {X 0,Y 279.241,Z 1181.365,A -85,B 0,C 180,E1 12483.179,E2 12483.179} C_VEL
LIN {X 0,Y 285.086,Z 1172.786,A -85,B 0,C 180,E1 12477.701,E2 12477.701} C_VEL
LIN {X 0,Y 292.689,Z 1162.518,A -85,B 0,C 180,E1 12472.546,E2 12472.546} C_VEL
LIN {X 0,Y 301.468,Z 1150.989,A -85,B 0,C 180,E1 12467.932,E2 12467.932} C_VEL
LIN {X 0,Y 311.391,Z 1138.026,A -85,B 0,C 180,E1 12463.738,E2 12463.738} C_VEL
LIN {X 0,Y 322.12,Z 1123.542,A -85,B 0,C 180,E1 12459.938,E2 12459.938} C_VEL
LIN {X 0,Y 333.413,Z 1107.635,A -85,B 0,C 180,E1 12456.511,E2 12456.511} C_VEL
LIN {X 0,Y 345.291,Z 1089.938,A -85,B 0,C 180,E1 12453.381,E2 12453.381} C_VEL
LIN {X 0,Y 357.103,Z 1071.044,A -85,B 0,C 180,E1 12450.637,E2 12450.637} C_VEL
LIN {X 0,Y 368.765,Z 1050.659,A -85,B 0,C 180,E1 12448.207,E2 12448.207} C_VEL
LIN {X 0,Y 379.785,Z 1029.506,A -85,B 0,C 180,E1 12446.13,E2 12446.13} C_VEL
LIN {X 0,Y 390.097,Z 1007.486,A -85,B 0,C 180,E1 12444.342,E2 12444.342} C_VEL
LIN {X 0,Y 399.508,Z 984.901,A -85,B 0,C 180,E1 12442.826,E2 12442.826} C_VEL
LIN {X 0,Y 407.923,Z 961.478,A -85,B 0,C 180,E1 12441.528,E2 12441.528} C_VEL
LIN {X 0,Y 418.532,Z 927.897,A -85,B 0,C 180,E1 12440.022,E2 12440.022} C_VEL
LIN {X 0,Y 428.948,Z 892.256,A -85,B 0,C 180,E1 12438.739,E2 12438.739} C_VEL
LIN {X 0,Y 429.746,Z 889.177,A -85,B 0,C 180,E1 12438.624,E2 12438.624} C_VEL
LIN {X 0,Y 419.03,Z 908.728,A -85,B 0,C 180,E1 12437.497,E2 12437.497} C_VEL
LIN {X 0,Y 415.746,Z 914.668,A -85,B 0,C 180,E1 12437.158,E2 12437.158} C_VEL
LIN {X 0,Y 408.135,Z 928.819,A -85,B 0,C 180,E1 12436.433,E2 12436.433} C_VEL
LIN {X 0,Y 400.119,Z 944.443,A -85,B 0,C 180,E1 12435.82,E2 12435.82} C_VEL
LIN {X 0,Y 391.597,Z 960.2,A -85,B 0,C 180,E1 12435.248,E2 12435.248} C_VEL
LIN {X 0,Y 386.328,Z 969.018,A -85,B 0,C 180,E1 12434.847,E2 12434.847} C_VEL
LIN {X 0,Y 378.059,Z 981.828,A -85,B 0,C 180,E1 12434.239,E2 12434.239} C_VEL
LIN {X 0,Y 368.118,Z 995.913,A -85,B 0,C 180,E1 12433.487,E2 12433.487} C_VEL
LIN {X 0,Y 357.535,Z 1009.488,A -85,B 0,C 180,E1 12432.6,E2 12432.6} C_VEL
LIN {X 0,Y 347.796,Z 1020.946,A -85,B 0,C 180,E1 12431.694,E2 12431.694} C_VEL
LIN {X 0,Y 338.96,Z 1030.577,A -85,B 0,C 180,E1 12430.787,E2 12430.787} C_VEL
LIN {X 0,Y 330.212,Z 1039.449,A -85,B 0,C 180,E1 12429.763,E2 12429.763} C_VEL
LIN {X 0,Y 322.649,Z 1046.725,A -85,B 0,C 180,E1 12428.734,E2 12428.734} C_VEL
LIN {X 0,Y 314.63,Z 1053.935,A -85,B 0,C 180,E1 12427.452,E2 12427.452} C_VEL
LIN {X 0,Y 308.506,Z 1059.243,A -85,B 0,C 180,E1 12426.327,E2 12426.327} C_VEL
LIN {X 0,Y 298.872,Z 1067.258,A -85,B 0,C 180,E1 12424.221,E2 12424.221} C_VEL
LIN {X 0,Y 293.3,Z 1071.687,A -85,B 0,C 180,E1 12422.697,E2 12422.697} C_VEL
LIN {X 0,Y 289.614,Z 1074.592,A -85,B 0,C 180,E1 12421.583,E2 12421.583} C_VEL
LIN {X 0,Y 288.97,Z 1075.309,A -85,B 0,C 180,E1 12421.289,E2 12421.289} C_VEL
LIN {X 0,Y 286.984,Z 1084.374,A -85,B 0,C 180,E1 12419.561,E2 12419.561} C_VEL
LIN {X 0,Y 285.111,Z 1091.921,A -85,B 0,C 180,E1 12417.789,E2 12417.789} C_VEL
LIN {X 0,Y 282.99,Z 1099.483,A -85,B 0,C 180,E1 12415.542,E2 12415.542} C_VEL
LIN {X 0,Y 280.927,Z 1105.576,A -85,B 0,C 180,E1 12413.049,E2 12413.049} C_VEL
LIN {X 0,Y 279.466,Z 1109.298,A -85,B 0,C 180,E1 12410.937,E2 12410.937} C_VEL
LIN {X 0,Y 278.255,Z 1111.861,A -85,B 0,C 180,E1 12408.811,E2 12408.811} C_VEL
LIN {X 0,Y 277.279,Z 1113.343,A -85,B 0,C 180,E1 12406.656,E2 12406.656} C_VEL
LIN {X 0,Y 276.544,Z 1113.757,A -85,B 0,C 180,E1 12404.481,E2 12404.481} C_VEL
LIN {X 0,Y 276.045,Z 1113.114,A -85,B 0,C 180,E1 12402.286,E2 12402.286} C_VEL
LIN {X 0,Y 275.762,Z 1111.211,A -85,B 0,C 180,E1 12399.908,E2 12399.908} C_VEL
LIN {X 0,Y 275.745,Z 1107.846,A -85,B 0,C 180,E1 12397.395,E2 12397.395} C_VEL
LIN {X 0,Y 276.094,Z 1101.932,A -85,B 0,C 180,E1 12394.471,E2 12394.471} C_VEL
LIN {X 0,Y 276.173,Z 1101.272,A -85,B 0,C 180,E1 12394.134,E2 12394.134} C_VEL
LIN {X 0,Y 277.865,Z 1101.933,A -85,B 0,C 180,E1 12392.806,E2 12392.806} C_VEL
LIN {X 0,Y 284.624,Z 1103.356,A -85,B 0,C 180,E1 12388.908,E2 12388.908} C_VEL
LIN {X 0,Y 295.557,Z 1104.163,A -85,B 0,C 180,E1 12384.654,E2 12384.654} C_VEL
LIN {X 0,Y 309.128,Z 1103.793,A -85,B 0,C 180,E1 12380.895,E2 12380.895} C_VEL
LIN {X 0,Y 319.063,Z 1102.975,A -85,B 0,C 180,E1 12378.777,E2 12378.777} C_VEL
LIN {X 0,Y 308.755,Z 1117.666,A -85,B 0,C 180,E1 12374.911,E2 12374.911} C_VEL
LIN {X 0,Y 299.362,Z 1130.958,A -85,B 0,C 180,E1 12370.643,E2 12370.643} C_VEL
LIN {X 0,Y 291.407,Z 1142.557,A -85,B 0,C 180,E1 12366.172,E2 12366.172} C_VEL
LIN {X 0,Y 284.694,Z 1152.76,A -85,B 0,C 180,E1 12361.321,E2 12361.321} C_VEL
LIN {X 0,Y 279.942,Z 1160.678,A -85,B 0,C 180,E1 12356.749,E2 12356.749} C_VEL
LIN {X 0,Y 275.95,Z 1168.278,A -85,B 0,C 180,E1 12351.247,E2 12351.247} C_VEL
LIN {X 0,Y 273.83,Z 1173.261,A -85,B 0,C 180,E1 12346.55,E2 12346.55} C_VEL
LIN {X 0,Y 272.65,Z 1177.041,A -85,B 0,C 180,E1 12341.854,E2 12341.854} C_VEL
LIN {X 0,Y 272.132,Z 1179.723,A -85,B 0,C 180,E1 12336.755,E2 12336.755} C_VEL
LIN {X 0,Y 272.012,Z 1180.816,A -85,B 0,C 180,E1 12332.531,E2 12332.531} C_VEL
LIN {X 0,Y 272.006,Z 1180.937,A -85,B 0,C 180,E1 12328.528,E2 12328.528} C_VEL
LIN {X 0,Y 272.063,Z 1180.221,A -85,B 0,C 180,E1 12324.731,E2 12324.731} C_VEL
LIN {X 0,Y 272.313,Z 1178.579,A -85,B 0,C 180,E1 12320.705,E2 12320.705} C_VEL
LIN {X 0,Y 272.964,Z 1175.876,A -85,B 0,C 180,E1 12316.444,E2 12316.444} C_VEL
LIN {X 0,Y 274.631,Z 1171.354,A -85,B 0,C 180,E1 12311.316,E2 12311.316} C_VEL
LIN {X 0,Y 277.52,Z 1165.118,A -85,B 0,C 180,E1 12306.204,E2 12306.204} C_VEL
LIN {X 0,Y 281.234,Z 1158.48,A -85,B 0,C 180,E1 12301.783,E2 12301.783} C_VEL
LIN {X 0,Y 287.453,Z 1148.503,A -85,B 0,C 180,E1 12296.426,E2 12296.426} C_VEL
LIN {X 0,Y 293.88,Z 1138.923,A -85,B 0,C 180,E1 12292.239,E2 12292.239} C_VEL
LIN {X 0,Y 302.713,Z 1126.291,A -85,B 0,C 180,E1 12287.64,E2 12287.64} C_VEL
LIN {X 0,Y 311.744,Z 1113.453,A -85,B 0,C 180,E1 12283.812,E2 12283.812} C_VEL
LIN {X 0,Y 322.436,Z 1098.264,A -85,B 0,C 180,E1 12280.012,E2 12280.012} C_VEL
LIN {X 0,Y 332.609,Z 1083.303,A -85,B 0,C 180,E1 12276.908,E2 12276.908} C_VEL
LIN {X 0,Y 343.692,Z 1066.561,A -85,B 0,C 180,E1 12273.958,E2 12273.958} C_VEL
LIN {X 0,Y 355.056,Z 1048.24,A -85,B 0,C 180,E1 12271.279,E2 12271.279} C_VEL
LIN {X 0,Y 367.171,Z 1027.455,A -85,B 0,C 180,E1 12268.737,E2 12268.737} C_VEL
LIN {X 0,Y 377.46,Z 1008.395,A -85,B 0,C 180,E1 12266.79,E2 12266.79} C_VEL
LIN {X 0,Y 388.473,Z 986.052,A -85,B 0,C 180,E1 12264.872,E2 12264.872} C_VEL
LIN {X 0,Y 397.623,Z 965.58,A -85,B 0,C 180,E1 12263.392,E2 12263.392} C_VEL
LIN {X 0,Y 398.812,Z 962.847,A -85,B 0,C 180,E1 12263.211,E2 12263.211} C_VEL
LIN {X 0,Y 401.044,Z 956.435,A -85,B 0,C 180,E1 12262.669,E2 12262.669} C_VEL
LIN {X 0,Y 405.018,Z 940.879,A -85,B 0,C 180,E1 12260.945,E2 12260.945} C_VEL
LIN {X 0,Y 407.049,Z 934.217,A -85,B 0,C 180,E1 12260.468,E2 12260.468} C_VEL
LIN {X 0,Y 414.537,Z 911.649,A -85,B 0,C 180,E1 12259.426,E2 12259.426} C_VEL
LIN {X 0,Y 421.711,Z 886.339,A -85,B 0,C 180,E1 12258.465,E2 12258.465} C_VEL
LIN {X 0,Y 430.37,Z 849.326,A -85,B 0,C 180,E1 12257.368,E2 12257.368} C_VEL
LIN {X 0,Y 444.119,Z 787.425,A -85,B 0,C 180,E1 12255.959,E2 12255.959} C_VEL
LIN {X 0,Y 456.532,Z 724.658,A -85,B 0,C 180,E1 12254.706,E2 12254.706} C_VEL
LIN {X 0,Y 466.924,Z 663.928,A -85,B 0,C 180,E1 12253.623,E2 12253.623} C_VEL
LIN {X 0,Y 472.279,Z 627.275,A -85,B 0,C 180,E1 12253.004,E2 12253.004} C_VEL
LIN {X 0,Y 468.058,Z 626.085,A -85,B 0,C 180,E1 12250.089,E2 12250.089} C_VEL
LIN {X 0,Y 464.08,Z 627.948,A -85,B 0,C 180,E1 12246.557,E2 12246.557} C_VEL
LIN {X 0,Y 462.143,Z 630.684,A -85,B 0,C 180,E1 12244.094,E2 12244.094} C_VEL
LIN {X 0,Y 460.743,Z 635.349,A -85,B 0,C 180,E1 12241.244,E2 12241.244} C_VEL
LIN {X 0,Y 460.434,Z 637.46,A -85,B 0,C 180,E1 12240.373,E2 12240.373} C_VEL
LIN {X 0,Y 455.868,Z 671.376,A -85,B 0,C 180,E1 12237.863,E2 12237.863} C_VEL
LIN {X 0,Y 450.587,Z 713.455,A -85,B 0,C 180,E1 12234.852,E2 12234.852} C_VEL
LIN {X 0,Y 447.655,Z 740.194,A -85,B 0,C 180,E1 12232.668,E2 12232.668} C_VEL
LIN {X 0,Y 445.565,Z 765.28,A -85,B 0,C 180,E1 12230.327,E2 12230.327} C_VEL
LIN {X 0,Y 444.433,Z 791.723,A -85,B 0,C 180,E1 12227.512,E2 12227.512} C_VEL
LIN {X 0,Y 444.784,Z 816.122,A -85,B 0,C 180,E1 12224.55,E2 12224.55} C_VEL
LIN {X 0,Y 444.911,Z 820.021,A -85,B 0,C 180,E1 12224.077,E2 12224.077} C_VEL
LIN {X 0,Y 434.848,Z 860.646,A -85,B 0,C 180,E1 12223.158,E2 12223.158} C_VEL
LIN {X 0,Y 424.92,Z 896.48,A -85,B 0,C 180,E1 12222.138,E2 12222.138} C_VEL
LIN {X 0,Y 414.59,Z 931.006,A -85,B 0,C 180,E1 12220.887,E2 12220.887} C_VEL
LIN {X 0,Y 404.563,Z 962.026,A -85,B 0,C 180,E1 12219.499,E2 12219.499} C_VEL
LIN {X 0,Y 395.845,Z 985.451,A -85,B 0,C 180,E1 12218.203,E2 12218.203} C_VEL
LIN {X 0,Y 386.756,Z 1006.848,A -85,B 0,C 180,E1 12216.786,E2 12216.786} C_VEL
LIN {X 0,Y 376.675,Z 1027.828,A -85,B 0,C 180,E1 12215.103,E2 12215.103} C_VEL
LIN {X 0,Y 365.893,Z 1048.16,A -85,B 0,C 180,E1 12213.15,E2 12213.15} C_VEL
LIN {X 0,Y 355.294,Z 1066.381,A -85,B 0,C 180,E1 12211.049,E2 12211.049} C_VEL
LIN {X 0,Y 343.623,Z 1084.897,A -85,B 0,C 180,E1 12208.489,E2 12208.489} C_VEL
LIN {X 0,Y 331.953,Z 1102.135,A -85,B 0,C 180,E1 12205.617,E2 12205.617} C_VEL
LIN {X 0,Y 320.504,Z 1117.963,A -85,B 0,C 180,E1 12202.407,E2 12202.407} C_VEL
LIN {X 0,Y 309.147,Z 1132.896,A -85,B 0,C 180,E1 12198.715,E2 12198.715} C_VEL
LIN {X 0,Y 298.037,Z 1147.01,A -85,B 0,C 180,E1 12194.389,E2 12194.389} C_VEL
LIN {X 0,Y 288.909,Z 1158.503,A -85,B 0,C 180,E1 12190.067,E2 12190.067} C_VEL
LIN {X 0,Y 280.506,Z 1169.192,A -85,B 0,C 180,E1 12185.019,E2 12185.019} C_VEL
LIN {X 0,Y 273.932,Z 1177.968,A -85,B 0,C 180,E1 12179.76,E2 12179.76} C_VEL
LIN {X 0,Y 269.037,Z 1185.336,A -85,B 0,C 180,E1 12174.127,E2 12174.127} C_VEL
LIN {X 0,Y 265.962,Z 1190.985,A -85,B 0,C 180,E1 12168.406,E2 12168.406} C_VEL
LIN {X 0,Y 264.517,Z 1194.808,A -85,B 0,C 180,E1 12163.106,E2 12163.106} C_VEL
LIN {X 0,Y 264.049,Z 1197.17,A -85,B 0,C 180,E1 12158.051,E2 12158.051} C_VEL
LIN {X 0,Y 263.996,Z 1198.442,A -85,B 0,C 180,E1 12153.254,E2 12153.254} C_VEL
LIN {X 0,Y 264.008,Z 1198.59,A -85,B 0,C 180,E1 12148.695,E2 12148.695} C_VEL
LIN {X 0,Y 263.999,Z 1197.875,A -85,B 0,C 180,E1 12144.128,E2 12144.128} C_VEL
LIN {X 0,Y 264.228,Z 1195.952,A -85,B 0,C 180,E1 12139.091,E2 12139.091} C_VEL
LIN {X 0,Y 265.294,Z 1192.58,A -85,B 0,C 180,E1 12133.578,E2 12133.578} C_VEL
LIN {X 0,Y 267.8,Z 1187.468,A -85,B 0,C 180,E1 12127.815,E2 12127.815} C_VEL
LIN {X 0,Y 272.027,Z 1180.716,A -85,B 0,C 180,E1 12122.17,E2 12122.17} C_VEL
LIN {X 0,Y 278.201,Z 1172.145,A -85,B 0,C 180,E1 12116.637,E2 12116.637} C_VEL
LIN {X 0,Y 286.384,Z 1161.599,A -85,B 0,C 180,E1 12111.318,E2 12111.318} C_VEL
LIN {X 0,Y 295.664,Z 1149.967,A -85,B 0,C 180,E1 12106.643,E2 12106.643} C_VEL
LIN {X 0,Y 306.066,Z 1136.868,A -85,B 0,C 180,E1 12102.409,E2 12102.409} C_VEL
LIN {X 0,Y 317.258,Z 1122.255,A -85,B 0,C 180,E1 12098.589,E2 12098.589} C_VEL
LIN {X 0,Y 329.586,Z 1105.349,A -85,B 0,C 180,E1 12095.001,E2 12095.001} C_VEL
LIN {X 0,Y 341.725,Z 1087.653,A -85,B 0,C 180,E1 12091.944,E2 12091.944} C_VEL
LIN {X 0,Y 353.684,Z 1068.948,A -85,B 0,C 180,E1 12089.281,E2 12089.281} C_VEL
LIN {X 0,Y 365.195,Z 1049.222,A -85,B 0,C 180,E1 12086.972,E2 12086.972} C_VEL
LIN {X 0,Y 376.6,Z 1027.768,A -85,B 0,C 180,E1 12084.902,E2 12084.902} C_VEL
LIN {X 0,Y 387.431,Z 1005.058,A -85,B 0,C 180,E1 12083.097,E2 12083.097} C_VEL
LIN {X 0,Y 397.414,Z 981.292,A -85,B 0,C 180,E1 12081.551,E2 12081.551} C_VEL
LIN {X 0,Y 405.894,Z 957.764,A -85,B 0,C 180,E1 12080.302,E2 12080.302} C_VEL
LIN {X 0,Y 416.957,Z 922.835,A -85,B 0,C 180,E1 12078.8,E2 12078.8} C_VEL
LIN {X 0,Y 420.014,Z 912.844,A -85,B 0,C 180,E1 12078.427,E2 12078.427} C_VEL
LIN {X 0,Y 416.118,Z 919.814,A -85,B 0,C 180,E1 12078.058,E2 12078.058} C_VEL
LIN {X 0,Y 409.353,Z 932.114,A -85,B 0,C 180,E1 12077.45,E2 12077.45} C_VEL
LIN {X 0,Y 399.449,Z 950.949,A -85,B 0,C 180,E1 12076.769,E2 12076.769} C_VEL
LIN {X 0,Y 391.611,Z 964.779,A -85,B 0,C 180,E1 12076.251,E2 12076.251} C_VEL
LIN {X 0,Y 386.276,Z 973.455,A -85,B 0,C 180,E1 12075.89,E2 12075.89} C_VEL
LIN {X 0,Y 377.839,Z 986.016,A -85,B 0,C 180,E1 12075.289,E2 12075.289} C_VEL
LIN {X 0,Y 369.019,Z 998.234,A -85,B 0,C 180,E1 12074.684,E2 12074.684} C_VEL
LIN {X 0,Y 357.316,Z 1012.885,A -85,B 0,C 180,E1 12073.76,E2 12073.76} C_VEL
LIN {X 0,Y 347.141,Z 1024.504,A -85,B 0,C 180,E1 12072.871,E2 12072.871} C_VEL
LIN {X 0,Y 337.776,Z 1034.413,A -85,B 0,C 180,E1 12071.959,E2 12071.959} C_VEL
LIN {X 0,Y 329.006,Z 1043.059,A -85,B 0,C 180,E1 12070.99,E2 12070.99} C_VEL
LIN {X 0,Y 320.424,Z 1050.913,A -85,B 0,C 180,E1 12069.883,E2 12069.883} C_VEL
LIN {X 0,Y 312.354,Z 1057.944,A -85,B 0,C 180,E1 12068.653,E2 12068.653} C_VEL
LIN {X 0,Y 302.103,Z 1066.366,A -85,B 0,C 180,E1 12066.806,E2 12066.806} C_VEL
LIN {X 0,Y 290.637,Z 1075.219,A -85,B 0,C 180,E1 12064.143,E2 12064.143} C_VEL
LIN {X 0,Y 281.811,Z 1081.801,A -85,B 0,C 180,E1 12061.423,E2 12061.423} C_VEL
LIN {X 0,Y 280.884,Z 1082.528,A -85,B 0,C 180,E1 12061.02,E2 12061.02} C_VEL
LIN {X 0,Y 278.515,Z 1091.521,A -85,B 0,C 180,E1 12058.971,E2 12058.971} C_VEL
LIN {X 0,Y 276.563,Z 1098.055,A -85,B 0,C 180,E1 12057.099,E2 12057.099} C_VEL
LIN {X 0,Y 274.795,Z 1103.361,A -85,B 0,C 180,E1 12055.199,E2 12055.199} C_VEL
LIN {X 0,Y 273.006,Z 1108.05,A -85,B 0,C 180,E1 12053.012,E2 12053.012} C_VEL
LIN {X 0,Y 271.276,Z 1111.943,A -85,B 0,C 180,E1 12050.453,E2 12050.453} C_VEL
LIN {X 0,Y 269.66,Z 1114.451,A -85,B 0,C 180,E1 12047.363,E2 12047.363} C_VEL
LIN {X 0,Y 268.743,Z 1114.967,A -85,B 0,C 180,E1 12044.904,E2 12044.904} C_VEL
LIN {X 0,Y 268.177,Z 1114.334,A -85,B 0,C 180,E1 12042.646,E2 12042.646} C_VEL
LIN {X 0,Y 267.85,Z 1112.616,A -85,B 0,C 180,E1 12040.368,E2 12040.368} C_VEL
LIN {X 0,Y 267.768,Z 1109.775,A -85,B 0,C 180,E1 12038.073,E2 12038.073} C_VEL
LIN {X 0,Y 268,Z 1105.333,A -85,B 0,C 180,E1 12035.418,E2 12035.418} C_VEL
LIN {X 0,Y 269.509,Z 1105.988,A -85,B 0,C 180,E1 12034.037,E2 12034.037} C_VEL
LIN {X 0,Y 275.985,Z 1107.725,A -85,B 0,C 180,E1 12029.762,E2 12029.762} C_VEL
LIN {X 0,Y 285.23,Z 1108.609,A -85,B 0,C 180,E1 12025.639,E2 12025.639} C_VEL
LIN {X 0,Y 298.015,Z 1108.686,A -85,B 0,C 180,E1 12021.632,E2 12021.632} C_VEL
LIN {X 0,Y 310.226,Z 1108.073,A -85,B 0,C 180,E1 12018.748,E2 12018.748} C_VEL
LIN {X 0,Y 299.346,Z 1122.859,A -85,B 0,C 180,E1 12014.546,E2 12014.546} C_VEL
LIN {X 0,Y 289.626,Z 1136.111,A -85,B 0,C 180,E1 12009.954,E2 12009.954} C_VEL
LIN {X 0,Y 281.561,Z 1147.314,A -85,B 0,C 180,E1 12005.123,E2 12005.123} C_VEL
LIN {X 0,Y 275.168,Z 1156.92,A -85,B 0,C 180,E1 12000.099,E2 12000.099} C_VEL
LIN {X 0,Y 270.378,Z 1164.692,A -85,B 0,C 180,E1 11994.937,E2 11994.937} C_VEL
LIN {X 0,Y 267.341,Z 1170.527,A -85,B 0,C 180,E1 11990.129,E2 11990.129} C_VEL
LIN {X 0,Y 265.192,Z 1175.765,A -85,B 0,C 180,E1 11984.412,E2 11984.412} C_VEL
LIN {X 0,Y 264.378,Z 1178.684,A -85,B 0,C 180,E1 11979.802,E2 11979.802} C_VEL
LIN {X 0,Y 264.085,Z 1180.387,A -85,B 0,C 180,E1 11975.652,E2 11975.652} C_VEL
LIN {X 0,Y 264.011,Z 1181.167,A -85,B 0,C 180,E1 11971.739,E2 11971.739} C_VEL
LIN {X 0,Y 264.014,Z 1181.134,A -85,B 0,C 180,E1 11967.832,E2 11967.832} C_VEL
LIN {X 0,Y 264.101,Z 1180.287,A -85,B 0,C 180,E1 11963.918,E2 11963.918} C_VEL
LIN {X 0,Y 264.444,Z 1178.405,A -85,B 0,C 180,E1 11959.546,E2 11959.546} C_VEL
LIN {X 0,Y 265.615,Z 1174.641,A -85,B 0,C 180,E1 11954.053,E2 11954.053} C_VEL
LIN {X 0,Y 267.634,Z 1169.913,A -85,B 0,C 180,E1 11949.214,E2 11949.214} C_VEL
LIN {X 0,Y 270.654,Z 1164.257,A -85,B 0,C 180,E1 11944.628,E2 11944.628} C_VEL
LIN {X 0,Y 276.022,Z 1155.569,A -85,B 0,C 180,E1 11939.046,E2 11939.046} C_VEL
LIN {X 0,Y 282.063,Z 1146.661,A -85,B 0,C 180,E1 11934.457,E2 11934.457} C_VEL
LIN {X 0,Y 290.615,Z 1134.776,A -85,B 0,C 180,E1 11929.442,E2 11929.442} C_VEL
LIN {X 0,Y 299.195,Z 1123.114,A -85,B 0,C 180,E1 11925.432,E2 11925.432} C_VEL
LIN {X 0,Y 309.941,Z 1108.577,A -85,B 0,C 180,E1 11921.269,E2 11921.269} C_VEL
LIN {X 0,Y 320.384,Z 1094.086,A -85,B 0,C 180,E1 11917.858,E2 11917.858} C_VEL
LIN {X 0,Y 332.725,Z 1076.437,A -85,B 0,C 180,E1 11914.4,E2 11914.4} C_VEL
LIN {X 0,Y 343.432,Z 1060.345,A -85,B 0,C 180,E1 11911.778,E2 11911.778} C_VEL
LIN {X 0,Y 355.83,Z 1040.565,A -85,B 0,C 180,E1 11909.087,E2 11909.087} C_VEL
LIN {X 0,Y 366.783,Z 1021.846,A -85,B 0,C 180,E1 11906.952,E2 11906.952} C_VEL
LIN {X 0,Y 378.529,Z 999.872,A -85,B 0,C 180,E1 11904.863,E2 11904.863} C_VEL
LIN {X 0,Y 389.576,Z 977.087,A -85,B 0,C 180,E1 11903.062,E2 11903.062} C_VEL
LIN {X 0,Y 399.791,Z 953.269,A -85,B 0,C 180,E1 11901.512,E2 11901.512} C_VEL
LIN {X 0,Y 407.049,Z 934.217,A -85,B 0,C 180,E1 11900.468,E2 11900.468} C_VEL
LIN {X 0,Y 409.051,Z 927.466,A -85,B 0,C 180,E1 11900.005,E2 11900.005} C_VEL
LIN {X 0,Y 412.818,Z 910.096,A -85,B 0,C 180,E1 11898.387,E2 11898.387} C_VEL
LIN {X 0,Y 414.365,Z 904.118,A -85,B 0,C 180,E1 11898.049,E2 11898.049} C_VEL
LIN {X 0,Y 421.02,Z 879.412,A -85,B 0,C 180,E1 11897.188,E2 11897.188} C_VEL
LIN {X 0,Y 431.082,Z 836.707,A -85,B 0,C 180,E1 11896.028,E2 11896.028} C_VEL
LIN {X 0,Y 445.117,Z 773.423,A -85,B 0,C 180,E1 11894.663,E2 11894.663} C_VEL
LIN {X 0,Y 456.914,Z 713.08,A -85,B 0,C 180,E1 11893.508,E2 11893.508} C_VEL
LIN {X 0,Y 466.568,Z 655.632,A -85,B 0,C 180,E1 11892.518,E2 11892.518} C_VEL
LIN {X 0,Y 469.664,Z 634.678,A -85,B 0,C 180,E1 11892.167,E2 11892.167} C_VEL
LIN {X 0,Y 466.483,Z 634.138,A -85,B 0,C 180,E1 11889.874,E2 11889.874} C_VEL
LIN {X 0,Y 462.881,Z 635.938,A -85,B 0,C 180,E1 11886.574,E2 11886.574} C_VEL
LIN {X 0,Y 461.014,Z 638.54,A -85,B 0,C 180,E1 11884.229,E2 11884.229} C_VEL
LIN {X 0,Y 459.587,Z 643.129,A -85,B 0,C 180,E1 11881.434,E2 11881.434} C_VEL
LIN {X 0,Y 459.392,Z 644.33,A -85,B 0,C 180,E1 11881.013,E2 11881.013} C_VEL
LIN {X 0,Y 454.554,Z 677.501,A -85,B 0,C 180,E1 11878.582,E2 11878.582} C_VEL
LIN {X 0,Y 448.854,Z 718.746,A -85,B 0,C 180,E1 11875.616,E2 11875.616} C_VEL
LIN {X 0,Y 445.589,Z 745.969,A -85,B 0,C 180,E1 11873.364,E2 11873.364} C_VEL
LIN {X 0,Y 443.151,Z 771.455,A -85,B 0,C 180,E1 11870.962,E2 11870.962} C_VEL
LIN {X 0,Y 441.65,Z 798.673,A -85,B 0,C 180,E1 11868.011,E2 11868.011} C_VEL
LIN {X 0,Y 441.698,Z 822.303,A -85,B 0,C 180,E1 11865.095,E2 11865.095} C_VEL
LIN {X 0,Y 441.585,Z 823.599,A -85,B 0,C 180,E1 11864.987,E2 11864.987} C_VEL
LIN {X 0,Y 429.886,Z 869.21,A -85,B 0,C 180,E1 11863.947,E2 11863.947} C_VEL
LIN {X 0,Y 419.539,Z 905.263,A -85,B 0,C 180,E1 11862.874,E2 11862.874} C_VEL
LIN {X 0,Y 408.893,Z 939.637,A -85,B 0,C 180,E1 11861.578,E2 11861.578} C_VEL
LIN {X 0,Y 400.167,Z 965.732,A -85,B 0,C 180,E1 11860.383,E2 11860.383} C_VEL
LIN {X 0,Y 391.306,Z 988.323,A -85,B 0,C 180,E1 11859.105,E2 11859.105} C_VEL
LIN {X 0,Y 381.259,Z 1010.741,A -85,B 0,C 180,E1 11857.581,E2 11857.581} C_VEL
LIN {X 0,Y 370.837,Z 1031.687,A -85,B 0,C 180,E1 11855.87,E2 11855.87} C_VEL
LIN {X 0,Y 359.324,Z 1052.256,A -85,B 0,C 180,E1 11853.821,E2 11853.821} C_VEL
LIN {X 0,Y 347.215,Z 1072.031,A -85,B 0,C 180,E1 11851.435,E2 11851.435} C_VEL
LIN {X 0,Y 335.381,Z 1089.958,A -85,B 0,C 180,E1 11848.826,E2 11848.826} C_VEL
LIN {X 0,Y 323.577,Z 1106.444,A -85,B 0,C 180,E1 11845.904,E2 11845.904} C_VEL
LIN {X 0,Y 311.46,Z 1122.393,A -85,B 0,C 180,E1 11842.457,E2 11842.457} C_VEL
LIN {X 0,Y 300.333,Z 1136.45,A -85,B 0,C 180,E1 11838.761,E2 11838.761} C_VEL
LIN {X 0,Y 289.566,Z 1149.536,A -85,B 0,C 180,E1 11834.501,E2 11834.501} C_VEL
LIN {X 0,Y 280.196,Z 1160.723,A -85,B 0,C 180,E1 11829.962,E2 11829.962} C_VEL
LIN {X 0,Y 271.802,Z 1171.032,A -85,B 0,C 180,E1 11824.761,E2 11824.761} C_VEL
LIN {X 0,Y 265.316,Z 1179.497,A -85,B 0,C 180,E1 11819.332,E2 11819.332} C_VEL
LIN {X 0,Y 260.52,Z 1186.557,A -85,B 0,C 180,E1 11813.465,E2 11813.465} C_VEL
LIN {X 0,Y 257.66,Z 1191.76,A -85,B 0,C 180,E1 11807.616,E2 11807.616} C_VEL
LIN {X 0,Y 256.338,Z 1195.335,A -85,B 0,C 180,E1 11801.928,E2 11801.928} C_VEL
LIN {X 0,Y 256.012,Z 1197.454,A -85,B 0,C 180,E1 11796.726,E2 11796.726} C_VEL
LIN {X 0,Y 256.006,Z 1198.28,A -85,B 0,C 180,E1 11792.012,E2 11792.012} C_VEL
LIN {X 0,Y 256.004,Z 1198.264,A -85,B 0,C 180,E1 11787.759,E2 11787.759} C_VEL
LIN {X 0,Y 256.021,Z 1197.29,A -85,B 0,C 180,E1 11782.818,E2 11782.818} C_VEL
LIN {X 0,Y 256.367,Z 1195.22,A -85,B 0,C 180,E1 11777.839,E2 11777.839} C_VEL
LIN {X 0,Y 257.739,Z 1191.563,A -85,B 0,C 180,E1 11772.15,E2 11772.15} C_VEL
LIN {X 0,Y 260.703,Z 1186.223,A -85,B 0,C 180,E1 11766.25,E2 11766.25} C_VEL
LIN {X 0,Y 265.549,Z 1179.171,A -85,B 0,C 180,E1 11760.436,E2 11760.436} C_VEL
LIN {X 0,Y 272.413,Z 1170.257,A -85,B 0,C 180,E1 11754.809,E2 11754.809} C_VEL
LIN {X 0,Y 281.023,Z 1159.72,A -85,B 0,C 180,E1 11749.59,E2 11749.59} C_VEL
LIN {X 0,Y 291.438,Z 1147.188,A -85,B 0,C 180,E1 11744.695,E2 11744.695} C_VEL
LIN {X 0,Y 302.932,Z 1133.123,A -85,B 0,C 180,E1 11740.312,E2 11740.312} C_VEL
LIN {X 0,Y 314.83,Z 1118.04,A -85,B 0,C 180,E1 11736.53,E2 11736.53} C_VEL
LIN {X 0,Y 327.243,Z 1101.375,A -85,B 0,C 180,E1 11733.151,E2 11733.151} C_VEL
LIN {X 0,Y 339.93,Z 1083.12,A -85,B 0,C 180,E1 11730.139,E2 11730.139} C_VEL
LIN {X 0,Y 352.098,Z 1064.174,A -85,B 0,C 180,E1 11727.574,E2 11727.574} C_VEL
LIN {X 0,Y 363.966,Z 1044.09,A -85,B 0,C 180,E1 11725.331,E2 11725.331} C_VEL
LIN {X 0,Y 375.204,Z 1022.972,A -85,B 0,C 180,E1 11723.396,E2 11723.396} C_VEL
LIN {X 0,Y 385.908,Z 1000.474,A -85,B 0,C 180,E1 11721.693,E2 11721.693} C_VEL
LIN {X 0,Y 395.563,Z 977.492,A -85,B 0,C 180,E1 11720.262,E2 11720.262} C_VEL
LIN {X 0,Y 404.113,Z 953.94,A -85,B 0,C 180,E1 11719.058,E2 11719.058} C_VEL
LIN {X 0,Y 409.21,Z 938.322,A -85,B 0,C 180,E1 11718.373,E2 11718.373} C_VEL
LIN {X 0,Y 400.682,Z 954.044,A -85,B 0,C 180,E1 11717.817,E2 11717.817} C_VEL
LIN {X 0,Y 392.756,Z 967.644,A -85,B 0,C 180,E1 11717.329,E2 11717.329} C_VEL
LIN {X 0,Y 386.193,Z 978.041,A -85,B 0,C 180,E1 11716.925,E2 11716.925} C_VEL
LIN {X 0,Y 371.193,Z 999.193,A -85,B 0,C 180,E1 11715.948,E2 11715.948} C_VEL
LIN {X 0,Y 357.245,Z 1016.281,A -85,B 0,C 180,E1 11714.922,E2 11714.922} C_VEL
LIN {X 0,Y 346.278,Z 1028.437,A -85,B 0,C 180,E1 11714.015,E2 11714.015} C_VEL
LIN {X 0,Y 337.222,Z 1037.709,A -85,B 0,C 180,E1 11713.198,E2 11713.198} C_VEL
LIN {X 0,Y 327.939,Z 1046.582,A -85,B 0,C 180,E1 11712.234,E2 11712.234} C_VEL
LIN {X 0,Y 318.33,Z 1055.102,A -85,B 0,C 180,E1 11711.046,E2 11711.046} C_VEL
LIN {X 0,Y 309.96,Z 1062.016,A -85,B 0,C 180,E1 11709.844,E2 11709.844} C_VEL
LIN {X 0,Y 299.557,Z 1070.2,A -85,B 0,C 180,E1 11708.059,E2 11708.059} C_VEL
LIN {X 0,Y 287.223,Z 1079.303,A -85,B 0,C 180,E1 11705.34,E2 11705.34} C_VEL
LIN {X 0,Y 277.22,Z 1086.33,A -85,B 0,C 180,E1 11702.396,E2 11702.396} C_VEL
LIN {X 0,Y 272.477,Z 1089.921,A -85,B 0,C 180,E1 11700.526,E2 11700.526} C_VEL
LIN {X 0,Y 269.715,Z 1098.652,A -85,B 0,C 180,E1 11698.088,E2 11698.088} C_VEL
LIN {X 0,Y 267.572,Z 1104.585,A -85,B 0,C 180,E1 11695.928,E2 11695.928} C_VEL
LIN {X 0,Y 265.607,Z 1109.318,A -85,B 0,C 180,E1 11693.653,E2 11693.653} C_VEL
LIN {X 0,Y 263.747,Z 1113.143,A -85,B 0,C 180,E1 11691.058,E2 11691.058} C_VEL
LIN {X 0,Y 261.978,Z 1115.663,A -85,B 0,C 180,E1 11687.882,E2 11687.882} C_VEL
LIN {X 0,Y 260.96,Z 1116.178,A -85,B 0,C 180,E1 11685.352,E2 11685.352} C_VEL
LIN {X 0,Y 260.318,Z 1115.55,A -85,B 0,C 180,E1 11683.027,E2 11683.027} C_VEL
LIN {X 0,Y 259.913,Z 1113.649,A -85,B 0,C 180,E1 11680.484,E2 11680.484} C_VEL
LIN {X 0,Y 259.816,Z 1110.331,A -85,B 0,C 180,E1 11677.843,E2 11677.843} C_VEL
LIN {X 0,Y 259.85,Z 1109.13,A -85,B 0,C 180,E1 11677.058,E2 11677.058} C_VEL
LIN {X 0,Y 261.093,Z 1109.915,A -85,B 0,C 180,E1 11675.569,E2 11675.569} C_VEL
LIN {X 0,Y 267.414,Z 1111.818,A -85,B 0,C 180,E1 11670.671,E2 11670.671} C_VEL
LIN {X 0,Y 276.501,Z 1113.002,A -85,B 0,C 180,E1 11666.158,E2 11666.158} C_VEL
LIN {X 0,Y 288.246,Z 1113.39,A -85,B 0,C 180,E1 11662.121,E2 11662.121} C_VEL
LIN {X 0,Y 301.514,Z 1112.814,A -85,B 0,C 180,E1 11658.768,E2 11658.768} C_VEL
LIN {X 0,Y 291.206,Z 1126.122,A -85,B 0,C 180,E1 11654.742,E2 11654.742} C_VEL
LIN {X 0,Y 280.65,Z 1139.87,A -85,B 0,C 180,E1 11649.626,E2 11649.626} C_VEL
LIN {X 0,Y 272.641,Z 1150.657,A -85,B 0,C 180,E1 11644.645,E2 11644.645} C_VEL
LIN {X 0,Y 266.134,Z 1159.948,A -85,B 0,C 180,E1 11639.239,E2 11639.239} C_VEL
LIN {X 0,Y 261.675,Z 1167.135,A -85,B 0,C 180,E1 11634.041,E2 11634.041} C_VEL
LIN {X 0,Y 258.48,Z 1173.225,A -85,B 0,C 180,E1 11628.263,E2 11628.263} C_VEL
LIN {X 0,Y 257.03,Z 1176.813,A -85,B 0,C 180,E1 11623.73,E2 11623.73} C_VEL
LIN {X 0,Y 256.328,Z 1179.394,A -85,B 0,C 180,E1 11619.206,E2 11619.206} C_VEL
LIN {X 0,Y 256.05,Z 1181.117,A -85,B 0,C 180,E1 11614.258,E2 11614.258} C_VEL
LIN {X 0,Y 256.009,Z 1181.554,A -85,B 0,C 180,E1 11609.331,E2 11609.331} C_VEL
LIN {X 0,Y 256.075,Z 1180.833,A -85,B 0,C 180,E1 11604.682,E2 11604.682} C_VEL
LIN {X 0,Y 256.361,Z 1179.225,A -85,B 0,C 180,E1 11600.348,E2 11600.348} C_VEL
LIN {X 0,Y 257.119,Z 1176.581,A -85,B 0,C 180,E1 11595.821,E2 11595.821} C_VEL
LIN {X 0,Y 259.046,Z 1172.12,A -85,B 0,C 180,E1 11590.36,E2 11590.36} C_VEL
LIN {X 0,Y 262.32,Z 1165.999,A -85,B 0,C 180,E1 11584.973,E2 11584.973} C_VEL
LIN {X 0,Y 266.497,Z 1159.433,A -85,B 0,C 180,E1 11580.317,E2 11580.317} C_VEL
LIN {X 0,Y 273.432,Z 1149.575,A -85,B 0,C 180,E1 11574.71,E2 11574.71} C_VEL
LIN {X 0,Y 280.556,Z 1140.031,A -85,B 0,C 180,E1 11570.338,E2 11570.338} C_VEL
LIN {X 0,Y 290.177,Z 1127.569,A -85,B 0,C 180,E1 11565.618,E2 11565.618} C_VEL
LIN {X 0,Y 299.969,Z 1114.855,A -85,B 0,C 180,E1 11561.702,E2 11561.702} C_VEL
LIN {X 0,Y 311.459,Z 1099.789,A -85,B 0,C 180,E1 11557.843,E2 11557.843} C_VEL
LIN {X 0,Y 322.334,Z 1084.983,A -85,B 0,C 180,E1 11554.716,E2 11554.716} C_VEL
LIN {X 0,Y 334.972,Z 1067.026,A -85,B 0,C 180,E1 11551.552,E2 11551.552} C_VEL
LIN {X 0,Y 346.631,Z 1049.414,A -85,B 0,C 180,E1 11548.987,E2 11548.987} C_VEL
LIN {X 0,Y 359.584,Z 1028.398,A -85,B 0,C 180,E1 11546.449,E2 11546.449} C_VEL
LIN {X 0,Y 371.536,Z 1007.362,A -85,B 0,C 180,E1 11544.347,E2 11544.347} C_VEL
LIN {X 0,Y 383.054,Z 984.733,A -85,B 0,C 180,E1 11542.481,E2 11542.481} C_VEL
LIN {X 0,Y 394.06,Z 960.426,A -85,B 0,C 180,E1 11540.833,E2 11540.833} C_VEL
LIN {X 0,Y 403.183,Z 937.715,A -85,B 0,C 180,E1 11539.55,E2 11539.55} C_VEL
LIN {X 0,Y 411.651,Z 912.96,A -85,B 0,C 180,E1 11538.407,E2 11538.407} C_VEL
LIN {X 0,Y 414.365,Z 904.118,A -85,B 0,C 180,E1 11538.049,E2 11538.049} C_VEL
LIN {X 0,Y 416.11,Z 897.094,A -85,B 0,C 180,E1 11537.658,E2 11537.658} C_VEL
LIN {X 0,Y 419.131,Z 878.894,A -85,B 0,C 180,E1 11536.216,E2 11536.216} C_VEL
LIN {X 0,Y 420.388,Z 872.726,A -85,B 0,C 180,E1 11535.929,E2 11535.929} C_VEL
LIN {X 0,Y 431.041,Z 828.278,A -85,B 0,C 180,E1 11534.796,E2 11534.796} C_VEL
LIN {X 0,Y 444.542,Z 767.774,A -85,B 0,C 180,E1 11533.539,E2 11533.539} C_VEL
LIN {X 0,Y 455.923,Z 709.934,A -85,B 0,C 180,E1 11532.462,E2 11532.462} C_VEL
LIN {X 0,Y 465.934,Z 650.116,A -85,B 0,C 180,E1 11531.458,E2 11531.458} C_VEL
LIN {X 0,Y 467.085,Z 642.223,A -85,B 0,C 180,E1 11531.317,E2 11531.317} C_VEL
LIN {X 0,Y 465.076,Z 642.118,A -85,B 0,C 180,E1 11529.779,E2 11529.779} C_VEL
LIN {X 0,Y 461.716,Z 643.77,A -85,B 0,C 180,E1 11526.716,E2 11526.716} C_VEL
LIN {X 0,Y 459.851,Z 646.39,A -85,B 0,C 180,E1 11524.365,E2 11524.365} C_VEL
LIN {X 0,Y 458.443,Z 650.782,A -85,B 0,C 180,E1 11521.687,E2 11521.687} C_VEL
LIN {X 0,Y 452.925,Z 685.716,A -85,B 0,C 180,E1 11519.149,E2 11519.149} C_VEL
LIN {X 0,Y 447.219,Z 724.023,A -85,B 0,C 180,E1 11516.387,E2 11516.387} C_VEL
LIN {X 0,Y 443.632,Z 750.834,A -85,B 0,C 180,E1 11514.146,E2 11514.146} C_VEL
LIN {X 0,Y 440.846,Z 775.75,A -85,B 0,C 180,E1 11511.785,E2 11511.785} C_VEL
LIN {X 0,Y 438.909,Z 802.865,A -85,B 0,C 180,E1 11508.835,E2 11508.835} C_VEL
LIN {X 0,Y 438.407,Z 826.71,A -85,B 0,C 180,E1 11505.917,E2 11505.917} C_VEL
LIN {X 0,Y 427.536,Z 868.483,A -85,B 0,C 180,E1 11504.983,E2 11504.983} C_VEL
LIN {X 0,Y 416.483,Z 906.521,A -85,B 0,C 180,E1 11503.874,E2 11503.874} C_VEL
LIN {X 0,Y 405.137,Z 942.479,A -85,B 0,C 180,E1 11502.525,E2 11502.525} C_VEL
LIN {X 0,Y 396.148,Z 968.144,A -85,B 0,C 180,E1 11501.336,E2 11501.336} C_VEL
LIN {X 0,Y 387.54,Z 989.593,A -85,B 0,C 180,E1 11500.127,E2 11500.127} C_VEL
LIN {X 0,Y 377.376,Z 1011.538,A -85,B 0,C 180,E1 11498.635,E2 11498.635} C_VEL
LIN {X 0,Y 366.069,Z 1033.328,A -85,B 0,C 180,E1 11496.838,E2 11496.838} C_VEL
LIN {X 0,Y 354.953,Z 1052.755,A -85,B 0,C 180,E1 11494.908,E2 11494.908} C_VEL
LIN {X 0,Y 342.902,Z 1071.844,A -85,B 0,C 180,E1 11492.606,E2 11492.606} C_VEL
LIN {X 0,Y 330.405,Z 1090.131,A -85,B 0,C 180,E1 11489.935,E2 11489.935} C_VEL
LIN {X 0,Y 318.767,Z 1105.97,A -85,B 0,C 180,E1 11487.135,E2 11487.135} C_VEL
LIN {X 0,Y 306.356,Z 1121.825,A -85,B 0,C 180,E1 11483.718,E2 11483.718} C_VEL
LIN {X 0,Y 294.341,Z 1136.407,A -85,B 0,C 180,E1 11479.843,E2 11479.843} C_VEL
LIN {X 0,Y 283.594,Z 1149.045,A -85,B 0,C 180,E1 11475.699,E2 11475.699} C_VEL
LIN {X 0,Y 273.773,Z 1160.293,A -85,B 0,C 180,E1 11471.098,E2 11471.098} C_VEL
LIN {X 0,Y 264.851,Z 1170.704,A -85,B 0,C 180,E1 11465.738,E2 11465.738} C_VEL
LIN {X 0,Y 258.022,Z 1179.166,A -85,B 0,C 180,E1 11460.211,E2 11460.211} C_VEL
LIN {X 0,Y 252.963,Z 1186.169,A -85,B 0,C 180,E1 11454.269,E2 11454.269} C_VEL
LIN {X 0,Y 249.915,Z 1191.265,A -85,B 0,C 180,E1 11448.422,E2 11448.422} C_VEL
LIN {X 0,Y 248.419,Z 1194.942,A -85,B 0,C 180,E1 11442.55,E2 11442.55} C_VEL
LIN {X 0,Y 248.035,Z 1197.033,A -85,B 0,C 180,E1 11437.39,E2 11437.39} C_VEL
LIN {X 0,Y 248.007,Z 1198,A -85,B 0,C 180,E1 11432.308,E2 11432.308} C_VEL
LIN {X 0,Y 248.009,Z 1198.016,A -85,B 0,C 180,E1 11427.918,E2 11427.918} C_VEL
LIN {X 0,Y 248.018,Z 1197.178,A -85,B 0,C 180,E1 11423.051,E2 11423.051} C_VEL
LIN {X 0,Y 248.386,Z 1195.047,A -85,B 0,C 180,E1 11417.678,E2 11417.678} C_VEL
LIN {X 0,Y 249.834,Z 1191.441,A -85,B 0,C 180,E1 11411.807,E2 11411.807} C_VEL
LIN {X 0,Y 252.966,Z 1186.142,A -85,B 0,C 180,E1 11405.725,E2 11405.725} C_VEL
LIN {X 0,Y 258.295,Z 1178.802,A -85,B 0,C 180,E1 11399.525,E2 11399.525} C_VEL
LIN {X 0,Y 265.585,Z 1169.839,A -85,B 0,C 180,E1 11393.764,E2 11393.764} C_VEL
LIN {X 0,Y 274.571,Z 1159.327,A -85,B 0,C 180,E1 11388.485,E2 11388.485} C_VEL
LIN {X 0,Y 285.447,Z 1146.793,A -85,B 0,C 180,E1 11383.52,E2 11383.52} C_VEL
LIN {X 0,Y 296.972,Z 1133.233,A -85,B 0,C 180,E1 11379.247,E2 11379.247} C_VEL
LIN {X 0,Y 309.265,Z 1118.166,A -85,B 0,C 180,E1 11375.435,E2 11375.435} C_VEL
LIN {X 0,Y 322.045,Z 1101.54,A -85,B 0,C 180,E1 11372.044,E2 11372.044} C_VEL
LIN {X 0,Y 335.076,Z 1083.36,A -85,B 0,C 180,E1 11369.031,E2 11369.031} C_VEL
LIN {X 0,Y 347.504,Z 1064.65,A -85,B 0,C 180,E1 11366.487,E2 11366.487} C_VEL
LIN {X 0,Y 359.241,Z 1045.315,A -85,B 0,C 180,E1 11364.327,E2 11364.327} C_VEL
LIN {X 0,Y 370.894,Z 1024.138,A -85,B 0,C 180,E1 11362.376,E2 11362.376} C_VEL
LIN {X 0,Y 381.689,Z 1002.29,A -85,B 0,C 180,E1 11360.711,E2 11360.711} C_VEL
LIN {X 0,Y 391.871,Z 978.865,A -85,B 0,C 180,E1 11359.248,E2 11359.248} C_VEL
LIN {X 0,Y 396.741,Z 966.266,A -85,B 0,C 180,E1 11358.568,E2 11358.568} C_VEL
LIN {X 0,Y 388.732,Z 978.795,A -85,B 0,C 180,E1 11358.091,E2 11358.091} C_VEL
LIN {X 0,Y 380.213,Z 991.023,A -85,B 0,C 180,E1 11357.574,E2 11357.574} C_VEL
LIN {X 0,Y 370.064,Z 1004.493,A -85,B 0,C 180,E1 11356.961,E2 11356.961} C_VEL
LIN {X 0,Y 357.317,Z 1019.676,A -85,B 0,C 180,E1 11356.083,E2 11356.083} C_VEL
LIN {X 0,Y 346.119,Z 1031.713,A -85,B 0,C 180,E1 11355.225,E2 11355.225} C_VEL
LIN {X 0,Y 333.655,Z 1044.023,A -85,B 0,C 180,E1 11354.157,E2 11354.157} C_VEL
LIN {X 0,Y 319.522,Z 1056.586,A -85,B 0,C 180,E1 11352.654,E2 11352.654} C_VEL
LIN {X 0,Y 307.677,Z 1066.107,A -85,B 0,C 180,E1 11351.048,E2 11351.048} C_VEL
LIN {X 0,Y 296.869,Z 1074.171,A -85,B 0,C 180,E1 11349.29,E2 11349.29} C_VEL
LIN {X 0,Y 284.295,Z 1083.031,A -85,B 0,C 180,E1 11346.665,E2 11346.665} C_VEL
LIN {X 0,Y 273.165,Z 1090.484,A -85,B 0,C 180,E1 11343.568,E2 11343.568} C_VEL
LIN {X 0,Y 264.388,Z 1096.223,A -85,B 0,C 180,E1 11340.217,E2 11340.217} C_VEL
LIN {X 0,Y 263.861,Z 1096.794,A -85,B 0,C 180,E1 11339.902,E2 11339.902} C_VEL
LIN {X 0,Y 260.863,Z 1104.835,A -85,B 0,C 180,E1 11337.144,E2 11337.144} C_VEL
LIN {X 0,Y 258.546,Z 1110.036,A -85,B 0,C 180,E1 11334.674,E2 11334.674} C_VEL
LIN {X 0,Y 256.734,Z 1113.51,A -85,B 0,C 180,E1 11332.391,E2 11332.391} C_VEL
LIN {X 0,Y 255.209,Z 1115.854,A -85,B 0,C 180,E1 11330.073,E2 11330.073} C_VEL
LIN {X 0,Y 253.867,Z 1117.207,A -85,B 0,C 180,E1 11327.489,E2 11327.489} C_VEL
LIN {X 0,Y 252.738,Z 1117.23,A -85,B 0,C 180,E1 11324.394,E2 11324.394} C_VEL
LIN {X 0,Y 252.058,Z 1115.291,A -85,B 0,C 180,E1 11321.257,E2 11321.257} C_VEL
LIN {X 0,Y 251.89,Z 1112.831,A -85,B 0,C 180,E1 11318.824,E2 11318.824} C_VEL
LIN {X 0,Y 256.368,Z 1115.102,A -85,B 0,C 180,E1 11313.601,E2 11313.601} C_VEL
LIN {X 0,Y 263.766,Z 1116.795,A -85,B 0,C 180,E1 11308.712,E2 11308.712} C_VEL
LIN {X 0,Y 273.35,Z 1117.592,A -85,B 0,C 180,E1 11304.436,E2 11304.436} C_VEL
LIN {X 0,Y 287.117,Z 1117.633,A -85,B 0,C 180,E1 11300.149,E2 11300.149} C_VEL
LIN {X 0,Y 292.573,Z 1117.564,A -85,B 0,C 180,E1 11298.731,E2 11298.731} C_VEL
LIN {X 0,Y 280.854,Z 1132.051,A -85,B 0,C 180,E1 11293.969,E2 11293.969} C_VEL
LIN {X 0,Y 271.938,Z 1143.161,A -85,B 0,C 180,E1 11289.452,E2 11289.452} C_VEL
LIN {X 0,Y 263.428,Z 1154.117,A -85,B 0,C 180,E1 11283.918,E2 11283.918} C_VEL
LIN {X 0,Y 257.55,Z 1162.255,A -85,B 0,C 180,E1 11278.78,E2 11278.78} C_VEL
LIN {X 0,Y 252.806,Z 1169.652,A -85,B 0,C 180,E1 11272.808,E2 11272.808} C_VEL
LIN {X 0,Y 250.236,Z 1174.507,A -85,B 0,C 180,E1 11267.681,E2 11267.681} C_VEL
LIN {X 0,Y 248.712,Z 1178.459,A -85,B 0,C 180,E1 11262.07,E2 11262.07} C_VEL
LIN {X 0,Y 248.147,Z 1180.721,A -85,B 0,C 180,E1 11256.713,E2 11256.713} C_VEL
LIN {X 0,Y 248.023,Z 1181.65,A -85,B 0,C 180,E1 11252.313,E2 11252.313} C_VEL
LIN {X 0,Y 248.02,Z 1181.727,A -85,B 0,C 180,E1 11248.386,E2 11248.386} C_VEL
LIN {X 0,Y 248.098,Z 1181.017,A -85,B 0,C 180,E1 11244.22,E2 11244.22} C_VEL
LIN {X 0,Y 248.426,Z 1179.388,A -85,B 0,C 180,E1 11239.802,E2 11239.802} C_VEL
LIN {X 0,Y 249.3,Z 1176.701,A -85,B 0,C 180,E1 11235.129,E2 11235.129} C_VEL
LIN {X 0,Y 251.561,Z 1171.949,A -85,B 0,C 180,E1 11229.286,E2 11229.286} C_VEL
LIN {X 0,Y 255.049,Z 1166.011,A -85,B 0,C 180,E1 11223.958,E2 11223.958} C_VEL
LIN {X 0,Y 260.068,Z 1158.747,A -85,B 0,C 180,E1 11218.736,E2 11218.736} C_VEL
LIN {X 0,Y 267.01,Z 1149.459,A -85,B 0,C 180,E1 11213.461,E2 11213.461} C_VEL
LIN {X 0,Y 274.529,Z 1139.966,A -85,B 0,C 180,E1 11209.039,E2 11209.039} C_VEL
LIN {X 0,Y 285.211,Z 1126.76,A -85,B 0,C 180,E1 11204.058,E2 11204.058} C_VEL
LIN {X 0,Y 295.015,Z 1114.624,A -85,B 0,C 180,E1 11200.312,E2 11200.312} C_VEL
LIN {X 0,Y 307.589,Z 1098.673,A -85,B 0,C 180,E1 11196.273,E2 11196.273} C_VEL
LIN {X 0,Y 320.168,Z 1082.181,A -85,B 0,C 180,E1 11192.856,E2 11192.856} C_VEL
LIN {X 0,Y 332.416,Z 1065.028,A -85,B 0,C 180,E1 11189.955,E2 11189.955} C_VEL
LIN {X 0,Y 345.34,Z 1045.983,A -85,B 0,C 180,E1 11187.273,E2 11187.273} C_VEL
LIN {X 0,Y 357.78,Z 1025.997,A -85,B 0,C 180,E1 11184.961,E2 11184.961} C_VEL
LIN {X 0,Y 370.315,Z 1003.944,A -85,B 0,C 180,E1 11182.853,E2 11182.853} C_VEL
LIN {X 0,Y 381.574,Z 982.138,A -85,B 0,C 180,E1 11181.12,E2 11181.12} C_VEL
LIN {X 0,Y 392.163,Z 958.849,A -85,B 0,C 180,E1 11179.599,E2 11179.599} C_VEL
LIN {X 0,Y 401.8,Z 934.711,A -85,B 0,C 180,E1 11178.295,E2 11178.295} C_VEL
LIN {X 0,Y 409.873,Z 911.251,A -85,B 0,C 180,E1 11177.249,E2 11177.249} C_VEL
LIN {X 0,Y 416.834,Z 886.893,A -85,B 0,C 180,E1 11176.37,E2 11176.37} C_VEL
LIN {X 0,Y 420.388,Z 872.726,A -85,B 0,C 180,E1 11175.929,E2 11175.929} C_VEL
LIN {X 0,Y 421.867,Z 865.52,A -85,B 0,C 180,E1 11175.587,E2 11175.587} C_VEL
LIN {X 0,Y 424.718,Z 847.907,A -85,B 0,C 180,E1 11174.329,E2 11174.329} C_VEL
LIN {X 0,Y 426.236,Z 840.646,A -85,B 0,C 180,E1 11174.031,E2 11174.031} C_VEL
LIN {X 0,Y 440.227,Z 780.516,A -85,B 0,C 180,E1 11172.769,E2 11172.769} C_VEL
LIN {X 0,Y 452.559,Z 720.232,A -85,B 0,C 180,E1 11171.645,E2 11171.645} C_VEL
LIN {X 0,Y 462.393,Z 664.055,A -85,B 0,C 180,E1 11170.703,E2 11170.703} C_VEL
LIN {X 0,Y 464.616,Z 649.853,A -85,B 0,C 180,E1 11170.478,E2 11170.478} C_VEL
LIN {X 0,Y 460.56,Z 651.604,A -85,B 0,C 180,E1 11166.858,E2 11166.858} C_VEL
LIN {X 0,Y 458.637,Z 654.23,A -85,B 0,C 180,E1 11164.501,E2 11164.501} C_VEL
LIN {X 0,Y 457.377,Z 657.831,A -85,B 0,C 180,E1 11162.323,E2 11162.323} C_VEL
LIN {X 0,Y 451.545,Z 692.489,A -85,B 0,C 180,E1 11159.826,E2 11159.826} C_VEL
LIN {X 0,Y 445.942,Z 726.896,A -85,B 0,C 180,E1 11157.341,E2 11157.341} C_VEL
LIN {X 0,Y 441.889,Z 754.433,A -85,B 0,C 180,E1 11155.051,E2 11155.051} C_VEL
LIN {X 0,Y 438.745,Z 779.56,A -85,B 0,C 180,E1 11152.668,E2 11152.668} C_VEL
LIN {X 0,Y 436.304,Z 807.065,A -85,B 0,C 180,E1 11149.669,E2 11149.669} C_VEL
LIN {X 0,Y 435.368,Z 829.986,A -85,B 0,C 180,E1 11146.86,E2 11146.86} C_VEL
LIN {X 0,Y 424.205,Z 871.592,A -85,B 0,C 180,E1 11145.934,E2 11145.934} C_VEL
LIN {X 0,Y 413.188,Z 908.953,A -85,B 0,C 180,E1 11144.85,E2 11144.85} C_VEL
LIN {X 0,Y 401.996,Z 943.88,A -85,B 0,C 180,E1 11143.551,E2 11143.551} C_VEL
LIN {X 0,Y 393.677,Z 967.075,A -85,B 0,C 180,E1 11142.492,E2 11142.492} C_VEL
LIN {X 0,Y 384.369,Z 989.688,A -85,B 0,C 180,E1 11141.237,E2 11141.237} C_VEL
LIN {X 0,Y 374.443,Z 1010.599,A -85,B 0,C 180,E1 11139.836,E2 11139.836} C_VEL
LIN {X 0,Y 362.899,Z 1032.463,A -85,B 0,C 180,E1 11138.066,E2 11138.066} C_VEL
LIN {X 0,Y 351.087,Z 1052.656,A -85,B 0,C 180,E1 11136.086,E2 11136.086} C_VEL
LIN {X 0,Y 338.736,Z 1071.635,A -85,B 0,C 180,E1 11133.806,E2 11133.806} C_VEL
LIN {X 0,Y 325.563,Z 1090.37,A -85,B 0,C 180,E1 11131.076,E2 11131.076} C_VEL
LIN {X 0,Y 313.099,Z 1106.863,A -85,B 0,C 180,E1 11128.149,E2 11128.149} C_VEL
LIN {X 0,Y 300.813,Z 1121.922,A -85,B 0,C 180,E1 11124.849,E2 11124.849} C_VEL
LIN {X 0,Y 287.866,Z 1137.09,A -85,B 0,C 180,E1 11120.762,E2 11120.762} C_VEL
LIN {X 0,Y 276.313,Z 1150.107,A -85,B 0,C 180,E1 11116.359,E2 11116.359} C_VEL
LIN {X 0,Y 265.844,Z 1161.68,A -85,B 0,C 180,E1 11111.446,E2 11111.446} C_VEL
LIN {X 0,Y 256.851,Z 1171.699,A -85,B 0,C 180,E1 11105.999,E2 11105.999} C_VEL
LIN {X 0,Y 249.746,Z 1180.077,A -85,B 0,C 180,E1 11100.141,E2 11100.141} C_VEL
LIN {X 0,Y 244.612,Z 1186.95,A -85,B 0,C 180,E1 11093.867,E2 11093.867} C_VEL
LIN {X 0,Y 241.6,Z 1192.019,A -85,B 0,C 180,E1 11087.582,E2 11087.582} C_VEL
LIN {X 0,Y 240.313,Z 1195.226,A -85,B 0,C 180,E1 11081.761,E2 11081.761} C_VEL
LIN {X 0,Y 240.012,Z 1197.118,A -85,B 0,C 180,E1 11076.215,E2 11076.215} C_VEL
LIN {X 0,Y 240.019,Z 1197.801,A -85,B 0,C 180,E1 11071.429,E2 11071.429} C_VEL
LIN {X 0,Y 240.005,Z 1197.668,A -85,B 0,C 180,E1 11066.653,E2 11066.653} C_VEL
LIN {X 0,Y 240.066,Z 1196.508,A -85,B 0,C 180,E1 11061.615,E2 11061.615} C_VEL
LIN {X 0,Y 240.648,Z 1194.184,A -85,B 0,C 180,E1 11056.052,E2 11056.052} C_VEL
LIN {X 0,Y 242.528,Z 1190.219,A -85,B 0,C 180,E1 11049.987,E2 11049.987} C_VEL
LIN {X 0,Y 246.482,Z 1184.287,A -85,B 0,C 180,E1 11043.495,E2 11043.495} C_VEL
LIN {X 0,Y 252.427,Z 1176.827,A -85,B 0,C 180,E1 11037.401,E2 11037.401} C_VEL
LIN {X 0,Y 260.565,Z 1167.493,A -85,B 0,C 180,E1 11031.56,E2 11031.56} C_VEL
LIN {X 0,Y 270.437,Z 1156.561,A -85,B 0,C 180,E1 11026.256,E2 11026.256} C_VEL
LIN {X 0,Y 281.153,Z 1144.613,A -85,B 0,C 180,E1 11021.68,E2 11021.68} C_VEL
LIN {X 0,Y 293.915,Z 1130.049,A -85,B 0,C 180,E1 11017.242,E2 11017.242} C_VEL
LIN {X 0,Y 306.863,Z 1114.548,A -85,B 0,C 180,E1 11013.469,E2 11013.469} C_VEL
LIN {X 0,Y 319.816,Z 1098.006,A -85,B 0,C 180,E1 11010.223,E2 11010.223} C_VEL
LIN {X 0,Y 333.113,Z 1079.734,A -85,B 0,C 180,E1 11007.313,E2 11007.313} C_VEL
LIN {X 0,Y 346.38,Z 1059.884,A -85,B 0,C 180,E1 11004.744,E2 11004.744} C_VEL
LIN {X 0,Y 358.959,Z 1039.24,A -85,B 0,C 180,E1 11002.568,E2 11002.568} C_VEL
LIN {X 0,Y 370.893,Z 1017.455,A -85,B 0,C 180,E1 11000.692,E2 11000.692} C_VEL
LIN {X 0,Y 381.969,Z 994.667,A -85,B 0,C 180,E1 10999.088,E2 10999.088} C_VEL
LIN {X 0,Y 383.674,Z 990.814,A -85,B 0,C 180,E1 10998.831,E2 10998.831} C_VEL
LIN {X 0,Y 370.204,Z 1008.279,A -85,B 0,C 180,E1 10998.059,E2 10998.059} C_VEL
LIN {X 0,Y 357.475,Z 1023.035,A -85,B 0,C 180,E1 10997.247,E2 10997.247} C_VEL
LIN {X 0,Y 346.126,Z 1034.901,A -85,B 0,C 180,E1 10996.443,E2 10996.443} C_VEL
LIN {X 0,Y 335.889,Z 1044.814,A -85,B 0,C 180,E1 10995.628,E2 10995.628} C_VEL
LIN {X 0,Y 325.601,Z 1054.066,A -85,B 0,C 180,E1 10994.68,E2 10994.68} C_VEL
LIN {X 0,Y 315.419,Z 1062.478,A -85,B 0,C 180,E1 10993.567,E2 10993.567} C_VEL
LIN {X 0,Y 305.525,Z 1070.089,A -85,B 0,C 180,E1 10992.282,E2 10992.282} C_VEL
LIN {X 0,Y 293.519,Z 1078.73,A -85,B 0,C 180,E1 10990.402,E2 10990.402} C_VEL
LIN {X 0,Y 279.702,Z 1087.933,A -85,B 0,C 180,E1 10987.601,E2 10987.601} C_VEL
LIN {X 0,Y 268.278,Z 1095.116,A -85,B 0,C 180,E1 10984.489,E2 10984.489} C_VEL
LIN {X 0,Y 259.022,Z 1100.81,A -85,B 0,C 180,E1 10981.041,E2 10981.041} C_VEL
LIN {X 0,Y 254.918,Z 1103.599,A -85,B 0,C 180,E1 10978.989,E2 10978.989} C_VEL
LIN {X 0,Y 251.737,Z 1110.555,A -85,B 0,C 180,E1 10975.9,E2 10975.9} C_VEL
LIN {X 0,Y 249.515,Z 1114.495,A -85,B 0,C 180,E1 10973.326,E2 10973.326} C_VEL
LIN {X 0,Y 247.82,Z 1116.932,A -85,B 0,C 180,E1 10970.947,E2 10970.947} C_VEL
LIN {X 0,Y 246.433,Z 1118.281,A -85,B 0,C 180,E1 10968.532,E2 10968.532} C_VEL
LIN {X 0,Y 245.258,Z 1118.564,A -85,B 0,C 180,E1 10965.841,E2 10965.841} C_VEL
LIN {X 0,Y 244.453,Z 1117.586,A -85,B 0,C 180,E1 10963.117,E2 10963.117} C_VEL
LIN {X 0,Y 244.099,Z 1116.146,A -85,B 0,C 180,E1 10961.119,E2 10961.119} C_VEL
LIN {X 0,Y 246.454,Z 1118.061,A -85,B 0,C 180,E1 10956.825,E2 10956.825} C_VEL
LIN {X 0,Y 252.013,Z 1120.107,A -85,B 0,C 180,E1 10951.568,E2 10951.568} C_VEL
LIN {X 0,Y 262.543,Z 1121.632,A -85,B 0,C 180,E1 10945.691,E2 10945.691} C_VEL
LIN {X 0,Y 275.998,Z 1122.088,A -85,B 0,C 180,E1 10940.922,E2 10940.922} C_VEL
LIN {X 0,Y 283.87,Z 1121.913,A -85,B 0,C 180,E1 10938.8,E2 10938.8} C_VEL
LIN {X 0,Y 272.692,Z 1135.058,A -85,B 0,C 180,E1 10934.164,E2 10934.164} C_VEL
LIN {X 0,Y 262.246,Z 1147.465,A -85,B 0,C 180,E1 10928.707,E2 10928.707} C_VEL
LIN {X 0,Y 254.779,Z 1156.712,A -85,B 0,C 180,E1 10923.601,E2 10923.601} C_VEL
LIN {X 0,Y 248.342,Z 1165.319,A -85,B 0,C 180,E1 10917.585,E2 10917.585} C_VEL
LIN {X 0,Y 244.48,Z 1171.145,A -85,B 0,C 180,E1 10912.359,E2 10912.359} C_VEL
LIN {X 0,Y 241.763,Z 1176.3,A -85,B 0,C 180,E1 10906.337,E2 10906.337} C_VEL
LIN {X 0,Y 240.52,Z 1179.499,A -85,B 0,C 180,E1 10900.785,E2 10900.785} C_VEL
LIN {X 0,Y 240.127,Z 1181.186,A -85,B 0,C 180,E1 10896.218,E2 10896.218} C_VEL
LIN {X 0,Y 240.024,Z 1181.958,A -85,B 0,C 180,E1 10891.913,E2 10891.913} C_VEL
LIN {X 0,Y 240.027,Z 1181.946,A -85,B 0,C 180,E1 10887.854,E2 10887.854} C_VEL
LIN {X 0,Y 240.136,Z 1181.149,A -85,B 0,C 180,E1 10883.548,E2 10883.548} C_VEL
LIN {X 0,Y 240.54,Z 1179.438,A -85,B 0,C 180,E1 10878.979,E2 10878.979} C_VEL
LIN {X 0,Y 241.894,Z 1176.061,A -85,B 0,C 180,E1 10873.184,E2 10873.184} C_VEL
LIN {X 0,Y 244.577,Z 1171.024,A -85,B 0,C 180,E1 10867.404,E2 10867.404} C_VEL
LIN {X 0,Y 248.474,Z 1165.161,A -85,B 0,C 180,E1 10862.177,E2 10862.177} C_VEL
LIN {X 0,Y 254.966,Z 1156.5,A -85,B 0,C 180,E1 10856.164,E2 10856.164} C_VEL
LIN {X 0,Y 261.768,Z 1148.097,A -85,B 0,C 180,E1 10851.497,E2 10851.497} C_VEL
LIN {X 0,Y 271.911,Z 1136.059,A -85,B 0,C 180,E1 10846.116,E2 10846.116} C_VEL
LIN {X 0,Y 281.425,Z 1124.83,A -85,B 0,C 180,E1 10842.054,E2 10842.054} C_VEL
LIN {X 0,Y 294.08,Z 1109.729,A -85,B 0,C 180,E1 10837.612,E2 10837.612} C_VEL
LIN {X 0,Y 305.754,Z 1095.373,A -85,B 0,C 180,E1 10834.176,E2 10834.176} C_VEL
LIN {X 0,Y 319.002,Z 1078.254,A -85,B 0,C 180,E1 10830.82,E2 10830.82} C_VEL
LIN {X 0,Y 332.046,Z 1060.517,A -85,B 0,C 180,E1 10827.961,E2 10827.961} C_VEL
LIN {X 0,Y 344.916,Z 1041.49,A -85,B 0,C 180,E1 10825.449,E2 10825.449} C_VEL
LIN {X 0,Y 358.076,Z 1020.411,A -85,B 0,C 180,E1 10823.151,E2 10823.151} C_VEL
LIN {X 0,Y 369.715,Z 999.968,A -85,B 0,C 180,E1 10821.307,E2 10821.307} C_VEL
LIN {X 0,Y 381.493,Z 976.883,A -85,B 0,C 180,E1 10819.584,E2 10819.584} C_VEL
LIN {X 0,Y 392.358,Z 952.725,A -85,B 0,C 180,E1 10818.101,E2 10818.101} C_VEL
LIN {X 0,Y 401.353,Z 929.699,A -85,B 0,C 180,E1 10816.94,E2 10816.94} C_VEL
LIN {X 0,Y 409.417,Z 905.47,A -85,B 0,C 180,E1 10815.934,E2 10815.934} C_VEL
LIN {X 0,Y 416.106,Z 881.721,A -85,B 0,C 180,E1 10815.127,E2 10815.127} C_VEL
LIN {X 0,Y 426.236,Z 840.646,A -85,B 0,C 180,E1 10814.031,E2 10814.031} C_VEL
LIN {X 0,Y 427.802,Z 833.349,A -85,B 0,C 180,E1 10813.741,E2 10813.741} C_VEL
LIN {X 0,Y 431.076,Z 814.479,A -85,B 0,C 180,E1 10812.513,E2 10812.513} C_VEL
LIN {X 0,Y 432.411,Z 808.185,A -85,B 0,C 180,E1 10812.287,E2 10812.287} C_VEL
LIN {X 0,Y 445.073,Z 751.02,A -85,B 0,C 180,E1 10811.184,E2 10811.184} C_VEL
LIN {X 0,Y 456.193,Z 693.567,A -85,B 0,C 180,E1 10810.192,E2 10810.192} C_VEL
LIN {X 0,Y 462.146,Z 658.022,A -85,B 0,C 180,E1 10809.621,E2 10809.621} C_VEL
LIN {X 0,Y 459.203,Z 659.562,A -85,B 0,C 180,E1 10806.878,E2 10806.878} C_VEL
LIN {X 0,Y 457.404,Z 662.067,A -85,B 0,C 180,E1 10804.639,E2 10804.639} C_VEL
LIN {X 0,Y 456.359,Z 664.878,A -85,B 0,C 180,E1 10802.967,E2 10802.967} C_VEL
LIN {X 0,Y 450.214,Z 698.823,A -85,B 0,C 180,E1 10800.541,E2 10800.541} C_VEL
LIN {X 0,Y 444.183,Z 733.81,A -85,B 0,C 180,E1 10797.996,E2 10797.996} C_VEL
LIN {X 0,Y 439.956,Z 760.184,A -85,B 0,C 180,E1 10795.764,E2 10795.764} C_VEL
LIN {X 0,Y 436.466,Z 785.192,A -85,B 0,C 180,E1 10793.373,E2 10793.373} C_VEL
LIN {X 0,Y 433.604,Z 812.522,A -85,B 0,C 180,E1 10790.359,E2 10790.359} C_VEL
LIN {X 0,Y 432.385,Z 833.302,A -85,B 0,C 180,E1 10787.813,E2 10787.813} C_VEL
LIN {X 0,Y 420.467,Z 876.897,A -85,B 0,C 180,E1 10786.847,E2 10786.847} C_VEL
LIN {X 0,Y 409.479,Z 913.085,A -85,B 0,C 180,E1 10785.783,E2 10785.783} C_VEL
LIN {X 0,Y 398.388,Z 946.977,A -85,B 0,C 180,E1 10784.522,E2 10784.522} C_VEL
LIN {X 0,Y 390.017,Z 969.406,A -85,B 0,C 180,E1 10783.492,E2 10783.492} C_VEL
LIN {X 0,Y 380.133,Z 992.367,A -85,B 0,C 180,E1 10782.203,E2 10782.203} C_VEL
LIN {X 0,Y 369.34,Z 1014.376,A -85,B 0,C 180,E1 10780.714,E2 10780.714} C_VEL
LIN {X 0,Y 358.313,Z 1034.304,A -85,B 0,C 180,E1 10779.072,E2 10779.072} C_VEL
LIN {X 0,Y 345.474,Z 1055.354,A -85,B 0,C 180,E1 10776.973,E2 10776.973} C_VEL
LIN {X 0,Y 332.647,Z 1074.525,A -85,B 0,C 180,E1 10774.639,E2 10774.639} C_VEL
LIN {X 0,Y 319.841,Z 1091.925,A -85,B 0,C 180,E1 10772.035,E2 10772.035} C_VEL
LIN {X 0,Y 306.084,Z 1109.351,A -85,B 0,C 180,E1 10768.851,E2 10768.851} C_VEL
LIN {X 0,Y 292.979,Z 1124.903,A -85,B 0,C 180,E1 10765.33,E2 10765.33} C_VEL
LIN {X 0,Y 280.379,Z 1138.977,A -85,B 0,C 180,E1 10761.347,E2 10761.347} C_VEL
LIN {X 0,Y 268.584,Z 1151.664,A -85,B 0,C 180,E1 10756.854,E2 10756.854} C_VEL
LIN {X 0,Y 257.921,Z 1162.933,A -85,B 0,C 180,E1 10751.816,E2 10751.816} C_VEL
LIN {X 0,Y 248.768,Z 1172.789,A -85,B 0,C 180,E1 10746.213,E2 10746.213} C_VEL
LIN {X 0,Y 241.467,Z 1181.038,A -85,B 0,C 180,E1 10740.065,E2 10740.065} C_VEL
LIN {X 0,Y 236.564,Z 1187.268,A -85,B 0,C 180,E1 10733.935,E2 10733.935} C_VEL
LIN {X 0,Y 233.463,Z 1192.287,A -85,B 0,C 180,E1 10727.238,E2 10727.238} C_VEL
LIN {X 0,Y 232.249,Z 1195.409,A -85,B 0,C 180,E1 10721.168,E2 10721.168} C_VEL
LIN {X 0,Y 232.01,Z 1196.996,A -85,B 0,C 180,E1 10715.686,E2 10715.686} C_VEL
LIN {X 0,Y 232.022,Z 1197.57,A -85,B 0,C 180,E1 10710.985,E2 10710.985} C_VEL
LIN {X 0,Y 232.004,Z 1197.335,A -85,B 0,C 180,E1 10706.043,E2 10706.043} C_VEL
LIN {X 0,Y 232.103,Z 1196.07,A -85,B 0,C 180,E1 10700.825,E2 10700.825} C_VEL
LIN {X 0,Y 232.908,Z 1193.499,A -85,B 0,C 180,E1 10694.816,E2 10694.816} C_VEL
LIN {X 0,Y 235.154,Z 1189.353,A -85,B 0,C 180,E1 10688.548,E2 10688.548} C_VEL
LIN {X 0,Y 239.457,Z 1183.432,A -85,B 0,C 180,E1 10682.114,E2 10682.114} C_VEL
LIN {X 0,Y 245.984,Z 1175.77,A -85,B 0,C 180,E1 10675.876,E2 10675.876} C_VEL
LIN {X 0,Y 254.395,Z 1166.662,A -85,B 0,C 180,E1 10670.156,E2 10670.156} C_VEL
LIN {X 0,Y 264.832,Z 1155.611,A -85,B 0,C 180,E1 10664.778,E2 10664.778} C_VEL
LIN {X 0,Y 276.643,Z 1142.985,A -85,B 0,C 180,E1 10659.979,E2 10659.979} C_VEL
LIN {X 0,Y 289.46,Z 1128.818,A -85,B 0,C 180,E1 10655.717,E2 10655.717} C_VEL
LIN {X 0,Y 302.885,Z 1113.151,A -85,B 0,C 180,E1 10651.958,E2 10651.958} C_VEL
LIN {X 0,Y 316.445,Z 1096.296,A -85,B 0,C 180,E1 10648.704,E2 10648.704} C_VEL
LIN {X 0,Y 330.021,Z 1077.998,A -85,B 0,C 180,E1 10645.86,E2 10645.86} C_VEL
LIN {X 0,Y 343.97,Z 1057.49,A -85,B 0,C 180,E1 10643.277,E2 10643.277} C_VEL
LIN {X 0,Y 356.452,Z 1037.371,A -85,B 0,C 180,E1 10641.215,E2 10641.215} C_VEL
LIN {X 0,Y 368.41,Z 1015.855,A -85,B 0,C 180,E1 10639.411,E2 10639.411} C_VEL
LIN {X 0,Y 370.263,Z 1012.325,A -85,B 0,C 180,E1 10639.14,E2 10639.14} C_VEL
LIN {X 0,Y 358.401,Z 1025.704,A -85,B 0,C 180,E1 10638.455,E2 10638.455} C_VEL
LIN {X 0,Y 346.222,Z 1038.166,A -85,B 0,C 180,E1 10637.652,E2 10637.652} C_VEL
LIN {X 0,Y 335.371,Z 1048.346,A -85,B 0,C 180,E1 10636.85,E2 10636.85} C_VEL
LIN {X 0,Y 324.517,Z 1057.764,A -85,B 0,C 180,E1 10635.916,E2 10635.916} C_VEL
LIN {X 0,Y 313.585,Z 1066.535,A -85,B 0,C 180,E1 10634.779,E2 10634.779} C_VEL
LIN {X 0,Y 303.388,Z 1074.073,A -85,B 0,C 180,E1 10633.525,E2 10633.525} C_VEL
LIN {X 0,Y 291.007,Z 1082.595,A -85,B 0,C 180,E1 10631.685,E2 10631.685} C_VEL
LIN {X 0,Y 276.71,Z 1091.676,A -85,B 0,C 180,E1 10628.939,E2 10628.939} C_VEL
LIN {X 0,Y 264.301,Z 1099.118,A -85,B 0,C 180,E1 10625.732,E2 10625.732} C_VEL
LIN {X 0,Y 254.157,Z 1105.02,A -85,B 0,C 180,E1 10622.139,E2 10622.139} C_VEL
LIN {X 0,Y 246.237,Z 1109.745,A -85,B 0,C 180,E1 10618.138,E2 10618.138} C_VEL
LIN {X 0,Y 245.243,Z 1110.811,A -85,B 0,C 180,E1 10617.352,E2 10617.352} C_VEL
LIN {X 0,Y 242.385,Z 1115.536,A -85,B 0,C 180,E1 10614.318,E2 10614.318} C_VEL
LIN {X 0,Y 240.331,Z 1118.211,A -85,B 0,C 180,E1 10611.627,E2 10611.627} C_VEL
LIN {X 0,Y 238.812,Z 1119.532,A -85,B 0,C 180,E1 10609.14,E2 10609.14} C_VEL
LIN {X 0,Y 237.512,Z 1119.788,A -85,B 0,C 180,E1 10606.364,E2 10606.364} C_VEL
LIN {X 0,Y 236.756,Z 1119.147,A -85,B 0,C 180,E1 10604.067,E2 10604.067} C_VEL
LIN {X 0,Y 238.334,Z 1121.512,A -85,B 0,C 180,E1 10598.851,E2 10598.851} C_VEL
LIN {X 0,Y 243.308,Z 1123.759,A -85,B 0,C 180,E1 10592.86,E2 10592.86} C_VEL
LIN {X 0,Y 251.523,Z 1125.358,A -85,B 0,C 180,E1 10587.438,E2 10587.438} C_VEL
LIN {X 0,Y 261.349,Z 1126.092,A -85,B 0,C 180,E1 10583.082,E2 10583.082} C_VEL
LIN {X 0,Y 275.033,Z 1126.106,A -85,B 0,C 180,E1 10578.815,E2 10578.815} C_VEL
LIN {X 0,Y 263.622,Z 1139.041,A -85,B 0,C 180,E1 10573.958,E2 10573.958} C_VEL
LIN {X 0,Y 253.951,Z 1149.946,A -85,B 0,C 180,E1 10568.761,E2 10568.761} C_VEL
LIN {X 0,Y 245.548,Z 1159.897,A -85,B 0,C 180,E1 10562.794,E2 10562.794} C_VEL
LIN {X 0,Y 239.965,Z 1167.054,A -85,B 0,C 180,E1 10557.283,E2 10557.283} C_VEL
LIN {X 0,Y 235.731,Z 1173.359,A -85,B 0,C 180,E1 10551.066,E2 10551.066} C_VEL
LIN {X 0,Y 233.468,Z 1177.491,A -85,B 0,C 180,E1 10545.401,E2 10545.401} C_VEL
LIN {X 0,Y 232.475,Z 1180.093,A -85,B 0,C 180,E1 10540.41,E2 10540.41} C_VEL
LIN {X 0,Y 232.108,Z 1181.653,A -85,B 0,C 180,E1 10535.661,E2 10535.661} C_VEL
LIN {X 0,Y 232.022,Z 1182.331,A -85,B 0,C 180,E1 10530.744,E2 10530.744} C_VEL
LIN {X 0,Y 232.07,Z 1182.005,A -85,B 0,C 180,E1 10525.555,E2 10525.555} C_VEL
LIN {X 0,Y 232.409,Z 1180.361,A -85,B 0,C 180,E1 10520.094,E2 10520.094} C_VEL
LIN {X 0,Y 233.306,Z 1177.868,A -85,B 0,C 180,E1 10515.103,E2 10515.103} C_VEL
LIN {X 0,Y 235.214,Z 1174.177,A -85,B 0,C 180,E1 10509.863,E2 10509.863} C_VEL
LIN {X 0,Y 239.283,Z 1168.036,A -85,B 0,C 180,E1 10503.445,E2 10503.445} C_VEL
LIN {X 0,Y 244.36,Z 1161.372,A -85,B 0,C 180,E1 10498.144,E2 10498.144} C_VEL
LIN {X 0,Y 251.7,Z 1152.681,A -85,B 0,C 180,E1 10492.574,E2 10492.574} C_VEL
LIN {X 0,Y 260.535,Z 1142.476,A -85,B 0,C 180,E1 10487.465,E2 10487.465} C_VEL
LIN {X 0,Y 270.911,Z 1130.956,A -85,B 0,C 180,E1 10482.742,E2 10482.742} C_VEL
LIN {X 0,Y 282.313,Z 1117.922,A -85,B 0,C 180,E1 10478.494,E2 10478.494} C_VEL
LIN {X 0,Y 294.415,Z 1103.986,A -85,B 0,C 180,E1 10474.732,E2 10474.732} C_VEL
LIN {X 0,Y 307.558,Z 1087.934,A -85,B 0,C 180,E1 10471.243,E2 10471.243} C_VEL
LIN {X 0,Y 321.97,Z 1069.415,A -85,B 0,C 180,E1 10467.965,E2 10467.965} C_VEL
LIN {X 0,Y 336.097,Z 1049.932,A -85,B 0,C 180,E1 10465.178,E2 10465.178} C_VEL
LIN {X 0,Y 349.356,Z 1029.879,A -85,B 0,C 180,E1 10462.847,E2 10462.847} C_VEL
LIN {X 0,Y 362.498,Z 1008.176,A -85,B 0,C 180,E1 10460.768,E2 10460.768} C_VEL
LIN {X 0,Y 374.71,Z 985.755,A -85,B 0,C 180,E1 10458.999,E2 10458.999} C_VEL
LIN {X 0,Y 385.396,Z 963.437,A -85,B 0,C 180,E1 10457.558,E2 10457.558} C_VEL
LIN {X 0,Y 395.207,Z 940.325,A -85,B 0,C 180,E1 10456.31,E2 10456.31} C_VEL
LIN {X 0,Y 403.278,Z 918.207,A -85,B 0,C 180,E1 10455.325,E2 10455.325} C_VEL
LIN {X 0,Y 410.883,Z 893.617,A -85,B 0,C 180,E1 10454.421,E2 10454.421} C_VEL
LIN {X 0,Y 419.979,Z 858.714,A -85,B 0,C 180,E1 10453.409,E2 10453.409} C_VEL
LIN {X 0,Y 432.398,Z 808.24,A -85,B 0,C 180,E1 10452.288,E2 10452.288} C_VEL
LIN {X 0,Y 432.411,Z 808.185,A -85,B 0,C 180,E1 10452.287,E2 10452.287} C_VEL
LIN {X 0,Y 433.94,Z 800.862,A -85,B 0,C 180,E1 10452.013,E2 10452.013} C_VEL
LIN {X 0,Y 437.257,Z 781.9,A -85,B 0,C 180,E1 10450.83,E2 10450.83} C_VEL
LIN {X 0,Y 438.508,Z 775.58,A -85,B 0,C 180,E1 10450.608,E2 10450.608} C_VEL
LIN {X 0,Y 449.625,Z 722.392,A -85,B 0,C 180,E1 10449.664,E2 10449.664} C_VEL
LIN {X 0,Y 459.124,Z 669.847,A -85,B 0,C 180,E1 10448.815,E2 10448.815} C_VEL
LIN {X 0,Y 459.727,Z 666.274,A -85,B 0,C 180,E1 10448.757,E2 10448.757} C_VEL
LIN {X 0,Y 457.84,Z 667.516,A -85,B 0,C 180,E1 10446.899,E2 10446.899} C_VEL
LIN {X 0,Y 456.107,Z 669.891,A -85,B 0,C 180,E1 10444.779,E2 10444.779} C_VEL
LIN {X 0,Y 455.286,Z 671.945,A -85,B 0,C 180,E1 10443.604,E2 10443.604} C_VEL
LIN {X 0,Y 448.303,Z 708.599,A -85,B 0,C 180,E1 10441.014,E2 10441.014} C_VEL
LIN {X 0,Y 442.556,Z 739.557,A -85,B 0,C 180,E1 10438.738,E2 10438.738} C_VEL
LIN {X 0,Y 437.961,Z 766.169,A -85,B 0,C 180,E1 10436.466,E2 10436.466} C_VEL
LIN {X 0,Y 434.079,Z 791.952,A -85,B 0,C 180,E1 10433.967,E2 10433.967} C_VEL
LIN {X 0,Y 430.924,Z 819.126,A -85,B 0,C 180,E1 10430.922,E2 10430.922} C_VEL
LIN {X 0,Y 429.543,Z 836.424,A -85,B 0,C 180,E1 10428.782,E2 10428.782} C_VEL
LIN {X 0,Y 418.525,Z 876.208,A -85,B 0,C 180,E1 10427.922,E2 10427.922} C_VEL
LIN {X 0,Y 407.103,Z 913.511,A -85,B 0,C 180,E1 10426.856,E2 10426.856} C_VEL
LIN {X 0,Y 395.837,Z 947.305,A -85,B 0,C 180,E1 10425.622,E2 10425.622} C_VEL
LIN {X 0,Y 387.369,Z 969.655,A -85,B 0,C 180,E1 10424.616,E2 10424.616} C_VEL
LIN {X 0,Y 377.665,Z 991.48,A -85,B 0,C 180,E1 10423.409,E2 10423.409} C_VEL
LIN {X 0,Y 366.93,Z 1013.057,A -85,B 0,C 180,E1 10421.986,E2 10421.986} C_VEL
LIN {X 0,Y 355.221,Z 1033.899,A -85,B 0,C 180,E1 10420.308,E2 10420.308} C_VEL
LIN {X 0,Y 342.673,Z 1053.948,A -85,B 0,C 180,E1 10418.339,E2 10418.339} C_VEL
LIN {X 0,Y 330.131,Z 1072.423,A -85,B 0,C 180,E1 10416.154,E2 10416.154} C_VEL
LIN {X 0,Y 316.905,Z 1090.073,A -85,B 0,C 180,E1 10413.584,E2 10413.584} C_VEL
LIN {X 0,Y 303.129,Z 1107.124,A -85,B 0,C 180,E1 10410.548,E2 10410.548} C_VEL
LIN {X 0,Y 290.11,Z 1122.246,A -85,B 0,C 180,E1 10407.236,E2 10407.236} C_VEL
LIN {X 0,Y 277.436,Z 1136.001,A -85,B 0,C 180,E1 10403.48,E2 10403.48} C_VEL
LIN {X 0,Y 264.555,Z 1149.448,A -85,B 0,C 180,E1 10398.88,E2 10398.88} C_VEL
LIN {X 0,Y 253.43,Z 1160.806,A -85,B 0,C 180,E1 10393.974,E2 10393.974} C_VEL
LIN {X 0,Y 243.442,Z 1170.901,A -85,B 0,C 180,E1 10388.326,E2 10388.326} C_VEL
LIN {X 0,Y 235.574,Z 1179.188,A -85,B 0,C 180,E1 10382.327,E2 10382.327} C_VEL
LIN {X 0,Y 229.702,Z 1186.059,A -85,B 0,C 180,E1 10375.8,E2 10375.8} C_VEL
LIN {X 0,Y 226.169,Z 1191.101,A -85,B 0,C 180,E1 10369.361,E2 10369.361} C_VEL
LIN {X 0,Y 224.494,Z 1194.43,A -85,B 0,C 180,E1 10363.126,E2 10363.126} C_VEL
LIN {X 0,Y 224.032,Z 1196.48,A -85,B 0,C 180,E1 10357.176,E2 10357.176} C_VEL
LIN {X 0,Y 224.022,Z 1197.242,A -85,B 0,C 180,E1 10352.043,E2 10352.043} C_VEL
LIN {X 0,Y 224.018,Z 1197.207,A -85,B 0,C 180,E1 10347.439,E2 10347.439} C_VEL
LIN {X 0,Y 224.054,Z 1196.29,A -85,B 0,C 180,E1 10342.045,E2 10342.045} C_VEL
LIN {X 0,Y 224.626,Z 1194.078,A -85,B 0,C 180,E1 10336.088,E2 10336.088} C_VEL
LIN {X 0,Y 226.608,Z 1190.344,A -85,B 0,C 180,E1 10329.596,E2 10329.596} C_VEL
LIN {X 0,Y 230.657,Z 1184.892,A -85,B 0,C 180,E1 10322.921,E2 10322.921} C_VEL
LIN {X 0,Y 236.978,Z 1177.668,A -85,B 0,C 180,E1 10316.442,E2 10316.442} C_VEL
LIN {X 0,Y 245.644,Z 1168.58,A -85,B 0,C 180,E1 10310.275,E2 10310.275} C_VEL
LIN {X 0,Y 256.595,Z 1157.482,A -85,B 0,C 180,E1 10304.509,E2 10304.509} C_VEL
LIN {X 0,Y 269.099,Z 1144.722,A -85,B 0,C 180,E1 10299.385,E2 10299.385} C_VEL
LIN {X 0,Y 282.267,Z 1130.812,A -85,B 0,C 180,E1 10295.02,E2 10295.02} C_VEL
LIN {X 0,Y 295.869,Z 1115.587,A -85,B 0,C 180,E1 10291.236,E2 10291.236} C_VEL
LIN {X 0,Y 309.961,Z 1098.706,A -85,B 0,C 180,E1 10287.882,E2 10287.882} C_VEL
LIN {X 0,Y 324.214,Z 1080.28,A -85,B 0,C 180,E1 10284.943,E2 10284.943} C_VEL
LIN {X 0,Y 337.665,Z 1061.388,A -85,B 0,C 180,E1 10282.495,E2 10282.495} C_VEL
LIN {X 0,Y 350.871,Z 1040.87,A -85,B 0,C 180,E1 10280.345,E2 10280.345} C_VEL
LIN {X 0,Y 356.506,Z 1031.402,A -85,B 0,C 180,E1 10279.478,E2 10279.478} C_VEL
LIN {X 0,Y 341.77,Z 1045.888,A -85,B 0,C 180,E1 10278.572,E2 10278.572} C_VEL
LIN {X 0,Y 325.482,Z 1059.944,A -85,B 0,C 180,E1 10277.337,E2 10277.337} C_VEL
LIN {X 0,Y 312.957,Z 1069.685,A -85,B 0,C 180,E1 10276.139,E2 10276.139} C_VEL
LIN {X 0,Y 301.439,Z 1077.957,A -85,B 0,C 180,E1 10274.798,E2 10274.798} C_VEL
LIN {X 0,Y 288.3,Z 1086.634,A -85,B 0,C 180,E1 10272.942,E2 10272.942} C_VEL
LIN {X 0,Y 273.29,Z 1095.701,A -85,B 0,C 180,E1 10270.191,E2 10270.191} C_VEL
LIN {X 0,Y 260.55,Z 1102.943,A -85,B 0,C 180,E1 10267.054,E2 10267.054} C_VEL
LIN {X 0,Y 249.399,Z 1109.046,A -85,B 0,C 180,E1 10263.316,E2 10263.316} C_VEL
LIN {X 0,Y 240.58,Z 1113.958,A -85,B 0,C 180,E1 10259.047,E2 10259.047} C_VEL
LIN {X 0,Y 234.719,Z 1117.612,A -85,B 0,C 180,E1 10254.622,E2 10254.622} C_VEL
LIN {X 0,Y 231.862,Z 1120.5,A -85,B 0,C 180,E1 10250.819,E2 10250.819} C_VEL
LIN {X 0,Y 230.185,Z 1121.873,A -85,B 0,C 180,E1 10247.456,E2 10247.456} C_VEL
LIN {X 0,Y 230.48,Z 1124.661,A -85,B 0,C 180,E1 10241.274,E2 10241.274} C_VEL
LIN {X 0,Y 234.55,Z 1127.237,A -85,B 0,C 180,E1 10234.496,E2 10234.496} C_VEL
LIN {X 0,Y 243.197,Z 1129.203,A -85,B 0,C 180,E1 10227.886,E2 10227.886} C_VEL
LIN {X 0,Y 254.264,Z 1130.076,A -85,B 0,C 180,E1 10222.727,E2 10222.727} C_VEL
LIN {X 0,Y 266.102,Z 1130.362,A -85,B 0,C 180,E1 10218.798,E2 10218.798} C_VEL
LIN {X 0,Y 254.507,Z 1142.699,A -85,B 0,C 180,E1 10213.749,E2 10213.749} C_VEL
LIN {X 0,Y 244.893,Z 1153.224,A -85,B 0,C 180,E1 10208.364,E2 10208.364} C_VEL
LIN {X 0,Y 236.859,Z 1162.223,A -85,B 0,C 180,E1 10202.404,E2 10202.404} C_VEL
LIN {X 0,Y 230.979,Z 1169.585,A -85,B 0,C 180,E1 10196.206,E2 10196.206} C_VEL
LIN {X 0,Y 227.204,Z 1174.966,A -85,B 0,C 180,E1 10190.079,E2 10190.079} C_VEL
LIN {X 0,Y 225.201,Z 1178.68,A -85,B 0,C 180,E1 10184.4,E2 10184.4} C_VEL
LIN {X 0,Y 224.264,Z 1181.336,A -85,B 0,C 180,E1 10178.19,E2 10178.19} C_VEL
LIN {X 0,Y 224.046,Z 1182.399,A -85,B 0,C 180,E1 10173.073,E2 10173.073} C_VEL
LIN {X 0,Y 224.032,Z 1182.538,A -85,B 0,C 180,E1 10168.469,E2 10168.469} C_VEL
LIN {X 0,Y 224.131,Z 1181.877,A -85,B 0,C 180,E1 10163.857,E2 10163.857} C_VEL
LIN {X 0,Y 224.518,Z 1180.413,A -85,B 0,C 180,E1 10159.223,E2 10159.223} C_VEL
LIN {X 0,Y 225.603,Z 1177.837,A -85,B 0,C 180,E1 10154.054,E2 10154.054} C_VEL
LIN {X 0,Y 228.22,Z 1173.502,A -85,B 0,C 180,E1 10147.869,E2 10147.869} C_VEL
LIN {X 0,Y 232.802,Z 1167.201,A -85,B 0,C 180,E1 10141.531,E2 10141.531} C_VEL
LIN {X 0,Y 239.124,Z 1159.722,A -85,B 0,C 180,E1 10135.637,E2 10135.637} C_VEL
LIN {X 0,Y 247.379,Z 1150.462,A -85,B 0,C 180,E1 10130.013,E2 10130.013} C_VEL
LIN {X 0,Y 257.096,Z 1140.103,A -85,B 0,C 180,E1 10124.946,E2 10124.946} C_VEL
LIN {X 0,Y 268.418,Z 1127.871,A -85,B 0,C 180,E1 10120.218,E2 10120.218} C_VEL
LIN {X 0,Y 280.688,Z 1114.608,A -85,B 0,C 180,E1 10116.042,E2 10116.042} C_VEL
LIN {X 0,Y 294.181,Z 1099.236,A -85,B 0,C 180,E1 10112.192,E2 10112.192} C_VEL
LIN {X 0,Y 309.037,Z 1081.474,A -85,B 0,C 180,E1 10108.611,E2 10108.611} C_VEL
LIN {X 0,Y 322.225,Z 1064.638,A -85,B 0,C 180,E1 10105.863,E2 10105.863} C_VEL
LIN {X 0,Y 336.304,Z 1045.225,A -85,B 0,C 180,E1 10103.269,E2 10103.269} C_VEL
LIN {X 0,Y 349.793,Z 1024.982,A -85,B 0,C 180,E1 10101.052,E2 10101.052} C_VEL
LIN {X 0,Y 362.104,Z 1004.514,A -85,B 0,C 180,E1 10099.208,E2 10099.208} C_VEL
LIN {X 0,Y 374.32,Z 981.908,A -85,B 0,C 180,E1 10097.527,E2 10097.527} C_VEL
LIN {X 0,Y 385.355,Z 959.028,A -85,B 0,C 180,E1 10096.119,E2 10096.119} C_VEL
LIN {X 0,Y 394.771,Z 936.269,A -85,B 0,C 180,E1 10094.972,E2 10094.972} C_VEL
LIN {X 0,Y 403.367,Z 912.322,A -85,B 0,C 180,E1 10093.969,E2 10093.969} C_VEL
LIN {X 0,Y 410.041,Z 890.188,A -85,B 0,C 180,E1 10093.212,E2 10093.212} C_VEL
LIN {X 0,Y 421.227,Z 847.513,A -85,B 0,C 180,E1 10092.057,E2 10092.057} C_VEL
LIN {X 0,Y 435.179,Z 790.229,A -85,B 0,C 180,E1 10090.887,E2 10090.887} C_VEL
LIN {X 0,Y 438.508,Z 775.58,A -85,B 0,C 180,E1 10090.608,E2 10090.608} C_VEL
LIN {X 0,Y 440.012,Z 768.229,A -85,B 0,C 180,E1 10090.344,E2 10090.344} C_VEL
LIN {X 0,Y 443.261,Z 749.179,A -85,B 0,C 180,E1 10089.199,E2 10089.199} C_VEL
LIN {X 0,Y 444.447,Z 742.839,A -85,B 0,C 180,E1 10088.99,E2 10088.99} C_VEL
LIN {X 0,Y 454.516,Z 690.985,A -85,B 0,C 180,E1 10088.145,E2 10088.145} C_VEL
LIN {X 0,Y 457.35,Z 674.638,A -85,B 0,C 180,E1 10087.876,E2 10087.876} C_VEL
LIN {X 0,Y 454.988,Z 677.359,A -85,B 0,C 180,E1 10085.17,E2 10085.17} C_VEL
LIN {X 0,Y 454.333,Z 678.843,A -85,B 0,C 180,E1 10084.271,E2 10084.271} C_VEL
LIN {X 0,Y 447.14,Z 714.113,A -85,B 0,C 180,E1 10081.794,E2 10081.794} C_VEL
LIN {X 0,Y 441.018,Z 745.463,A -85,B 0,C 180,E1 10079.471,E2 10079.471} C_VEL
LIN {X 0,Y 435.759,Z 773.813,A -85,B 0,C 180,E1 10077.024,E2 10077.024} C_VEL
LIN {X 0,Y 431.22,Z 801.871,A -85,B 0,C 180,E1 10074.223,E2 10074.223} C_VEL
LIN {X 0,Y 428.157,Z 825.667,A -85,B 0,C 180,E1 10071.489,E2 10071.489} C_VEL
LIN {X 0,Y 426.861,Z 839.701,A -85,B 0,C 180,E1 10069.764,E2 10069.764} C_VEL
LIN {X 0,Y 415.077,Z 880.948,A -85,B 0,C 180,E1 10068.871,E2 10068.871} C_VEL
LIN {X 0,Y 404.276,Z 915.633,A -85,B 0,C 180,E1 10067.886,E2 10067.886} C_VEL
LIN {X 0,Y 393.713,Z 946.961,A -85,B 0,C 180,E1 10066.766,E2 10066.766} C_VEL
LIN {X 0,Y 384.5,Z 970.523,A -85,B 0,C 180,E1 10065.719,E2 10065.719} C_VEL
LIN {X 0,Y 375.067,Z 991.377,A -85,B 0,C 180,E1 10064.588,E2 10064.588} C_VEL
LIN {X 0,Y 363.593,Z 1013.704,A -85,B 0,C 180,E1 10063.129,E2 10063.129} C_VEL
LIN {X 0,Y 351.671,Z 1034.549,A -85,B 0,C 180,E1 10061.473,E2 10061.473} C_VEL
LIN {X 0,Y 338.834,Z 1054.476,A -85,B 0,C 180,E1 10059.529,E2 10059.529} C_VEL
LIN {X 0,Y 324.965,Z 1074.095,A -85,B 0,C 180,E1 10057.189,E2 10057.189} C_VEL
LIN {X 0,Y 312.38,Z 1090.475,A -85,B 0,C 180,E1 10054.804,E2 10054.804} C_VEL
LIN {X 0,Y 298.329,Z 1107.344,A -85,B 0,C 180,E1 10051.798,E2 10051.798} C_VEL
LIN {X 0,Y 284.822,Z 1122.518,A -85,B 0,C 180,E1 10048.461,E2 10048.461} C_VEL
LIN {X 0,Y 271.875,Z 1136.083,A -85,B 0,C 180,E1 10044.727,E2 10044.727} C_VEL
LIN {X 0,Y 258.875,Z 1149.128,A -85,B 0,C 180,E1 10040.225,E2 10040.225} C_VEL
LIN {X 0,Y 247.362,Z 1160.405,A -85,B 0,C 180,E1 10035.304,E2 10035.304} C_VEL
LIN {X 0,Y 236.891,Z 1170.51,A -85,B 0,C 180,E1 10029.59,E2 10029.59} C_VEL
LIN {X 0,Y 228.54,Z 1178.82,A -85,B 0,C 180,E1 10023.45,E2 10023.45} C_VEL
LIN {X 0,Y 222.246,Z 1185.726,A -85,B 0,C 180,E1 10016.733,E2 10016.733} C_VEL
LIN {X 0,Y 218.415,Z 1190.799,A -85,B 0,C 180,E1 10010.077,E2 10010.077} C_VEL
LIN {X 0,Y 216.567,Z 1194.15,A -85,B 0,C 180,E1 10003.616,E2 10003.616} C_VEL
LIN {X 0,Y 216.045,Z 1196.209,A -85,B 0,C 180,E1 9997.442,E2 9997.442} C_VEL
LIN {X 0,Y 216.025,Z 1196.978,A -85,B 0,C 180,E1 9992.119,E2 9992.119} C_VEL
LIN {X 0,Y 216.02,Z 1196.944,A -85,B 0,C 180,E1 9987.344,E2 9987.344} C_VEL
LIN {X 0,Y 216.057,Z 1196.099,A -85,B 0,C 180,E1 9982.016,E2 9982.016} C_VEL
LIN {X 0,Y 216.689,Z 1193.847,A -85,B 0,C 180,E1 9975.703,E2 9975.703} C_VEL
LIN {X 0,Y 218.773,Z 1190.217,A -85,B 0,C 180,E1 9969.112,E2 9969.112} C_VEL
LIN {X 0,Y 222.855,Z 1185.028,A -85,B 0,C 180,E1 9962.472,E2 9962.472} C_VEL
LIN {X 0,Y 229.429,Z 1177.893,A -85,B 0,C 180,E1 9955.789,E2 9955.789} C_VEL
LIN {X 0,Y 238.429,Z 1168.923,A -85,B 0,C 180,E1 9949.454,E2 9949.454} C_VEL
LIN {X 0,Y 249.299,Z 1158.439,A -85,B 0,C 180,E1 9943.782,E2 9943.782} C_VEL
LIN {X 0,Y 261.585,Z 1146.455,A -85,B 0,C 180,E1 9938.757,E2 9938.757} C_VEL
LIN {X 0,Y 275.522,Z 1132.288,A -85,B 0,C 180,E1 9934.161,E2 9934.161} C_VEL
LIN {X 0,Y 289.78,Z 1116.935,A -85,B 0,C 180,E1 9930.25,E2 9930.25} C_VEL
LIN {X 0,Y 303.954,Z 1100.621,A -85,B 0,C 180,E1 9926.936,E2 9926.936} C_VEL
LIN {X 0,Y 318.124,Z 1083.053,A -85,B 0,C 180,E1 9924.064,E2 9924.064} C_VEL
LIN {X 0,Y 332.217,Z 1063.896,A -85,B 0,C 180,E1 9921.543,E2 9921.543} C_VEL
LIN {X 0,Y 342.665,Z 1048.482,A -85,B 0,C 180,E1 9919.839,E2 9919.839} C_VEL
LIN {X 0,Y 325.4,Z 1063.102,A -85,B 0,C 180,E1 9918.637,E2 9918.637} C_VEL
LIN {X 0,Y 311.341,Z 1073.673,A -85,B 0,C 180,E1 9917.378,E2 9917.378} C_VEL
LIN {X 0,Y 299.529,Z 1081.805,A -85,B 0,C 180,E1 9916.086,E2 9916.086} C_VEL
LIN {X 0,Y 285.753,Z 1090.567,A -85,B 0,C 180,E1 9914.236,E2 9914.236} C_VEL
LIN {X 0,Y 270.251,Z 1099.573,A -85,B 0,C 180,E1 9911.525,E2 9911.525} C_VEL
LIN {X 0,Y 256.467,Z 1106.964,A -85,B 0,C 180,E1 9908.294,E2 9908.294} C_VEL
LIN {X 0,Y 244.516,Z 1113.122,A -85,B 0,C 180,E1 9904.456,E2 9904.456} C_VEL
LIN {X 0,Y 234.901,Z 1118.041,A -85,B 0,C 180,E1 9900,E2 9900} C_VEL
LIN {X 0,Y 228.373,Z 1121.829,A -85,B 0,C 180,E1 9895.228,E2 9895.228} C_VEL
LIN {X 0,Y 224.169,Z 1125.172,A -85,B 0,C 180,E1 9889.463,E2 9889.463} C_VEL
LIN {X 0,Y 223.218,Z 1128.438,A -85,B 0,C 180,E1 9882.266,E2 9882.266} C_VEL
LIN {X 0,Y 229.138,Z 1131.747,A -85,B 0,C 180,E1 9872.73,E2 9872.73} C_VEL
LIN {X 0,Y 238.804,Z 1133.394,A -85,B 0,C 180,E1 9866.159,E2 9866.159} C_VEL
LIN {X 0,Y 249.27,Z 1134.091,A -85,B 0,C 180,E1 9861.556,E2 9861.556} C_VEL
LIN {X 0,Y 257.323,Z 1134.175,A -85,B 0,C 180,E1 9858.878,E2 9858.878} C_VEL
LIN {X 0,Y 245.861,Z 1145.874,A -85,B 0,C 180,E1 9853.742,E2 9853.742} C_VEL
LIN {X 0,Y 235.796,Z 1156.203,A -85,B 0,C 180,E1 9847.933,E2 9847.933} C_VEL
LIN {X 0,Y 228.488,Z 1164.148,A -85,B 0,C 180,E1 9842.271,E2 9842.271} C_VEL
LIN {X 0,Y 222.402,Z 1171.316,A -85,B 0,C 180,E1 9835.572,E2 9835.572} C_VEL
LIN {X 0,Y 219.026,Z 1176.021,A -85,B 0,C 180,E1 9829.747,E2 9829.747} C_VEL
LIN {X 0,Y 216.903,Z 1179.889,A -85,B 0,C 180,E1 9823.058,E2 9823.058} C_VEL
LIN {X 0,Y 216.212,Z 1181.858,A -85,B 0,C 180,E1 9817.443,E2 9817.443} C_VEL
LIN {X 0,Y 216.044,Z 1182.706,A -85,B 0,C 180,E1 9812.656,E2 9812.656} C_VEL
LIN {X 0,Y 216.038,Z 1182.779,A -85,B 0,C 180,E1 9808.147,E2 9808.147} C_VEL
LIN {X 0,Y 216.162,Z 1182.075,A -85,B 0,C 180,E1 9803.363,E2 9803.363} C_VEL
LIN {X 0,Y 216.616,Z 1180.575,A -85,B 0,C 180,E1 9798.555,E2 9798.555} C_VEL
LIN {X 0,Y 217.862,Z 1177.971,A -85,B 0,C 180,E1 9793.197,E2 9793.197} C_VEL
LIN {X 0,Y 220.943,Z 1173.329,A -85,B 0,C 180,E1 9786.535,E2 9786.535} C_VEL
LIN {X 0,Y 225.552,Z 1167.496,A -85,B 0,C 180,E1 9780.527,E2 9780.527} C_VEL
LIN {X 0,Y 232.42,Z 1159.946,A -85,B 0,C 180,E1 9774.4,E2 9774.4} C_VEL
LIN {X 0,Y 241.313,Z 1150.533,A -85,B 0,C 180,E1 9768.589,E2 9768.589} C_VEL
LIN {X 0,Y 251.772,Z 1140.006,A -85,B 0,C 180,E1 9763.389,E2 9763.389} C_VEL
LIN {X 0,Y 263.664,Z 1127.708,A -85,B 0,C 180,E1 9758.634,E2 9758.634} C_VEL
LIN {X 0,Y 277.262,Z 1113.503,A -85,B 0,C 180,E1 9754.235,E2 9754.235} C_VEL
LIN {X 0,Y 291.185,Z 1098.213,A -85,B 0,C 180,E1 9750.476,E2 9750.476} C_VEL
LIN {X 0,Y 305.632,Z 1081.356,A -85,B 0,C 180,E1 9747.151,E2 9747.151} C_VEL
LIN {X 0,Y 319.959,Z 1063.6,A -85,B 0,C 180,E1 9744.305,E2 9744.305} C_VEL
LIN {X 0,Y 334.43,Z 1043.944,A -85,B 0,C 180,E1 9741.761,E2 9741.761} C_VEL
LIN {X 0,Y 348.545,Z 1022.927,A -85,B 0,C 180,E1 9739.553,E2 9739.553} C_VEL
LIN {X 0,Y 361.171,Z 1002.32,A -85,B 0,C 180,E1 9737.767,E2 9737.767} C_VEL
LIN {X 0,Y 372.383,Z 981.591,A -85,B 0,C 180,E1 9736.285,E2 9736.285} C_VEL
LIN {X 0,Y 383.029,Z 959.847,A -85,B 0,C 180,E1 9734.977,E2 9734.977} C_VEL
LIN {X 0,Y 392.399,Z 937.738,A -85,B 0,C 180,E1 9733.881,E2 9733.881} C_VEL
LIN {X 0,Y 401.5,Z 912.722,A -85,B 0,C 180,E1 9732.854,E2 9732.854} C_VEL
LIN {X 0,Y 407.68,Z 892.544,A -85,B 0,C 180,E1 9732.177,E2 9732.177} C_VEL
LIN {X 0,Y 419.038,Z 850.418,A -85,B 0,C 180,E1 9731.043,E2 9731.043} C_VEL
LIN {X 0,Y 432.939,Z 794.6,A -85,B 0,C 180,E1 9729.921,E2 9729.921} C_VEL
LIN {X 0,Y 444.367,Z 743.213,A -85,B 0,C 180,E1 9728.996,E2 9728.996} C_VEL
LIN {X 0,Y 444.447,Z 742.839,A -85,B 0,C 180,E1 9728.99,E2 9728.99} C_VEL
LIN {X 0,Y 445.907,Z 735.462,A -85,B 0,C 180,E1 9728.74,E2 9728.74} C_VEL
LIN {X 0,Y 449.017,Z 716.321,A -85,B 0,C 180,E1 9727.629,E2 9727.629} C_VEL
LIN {X 0,Y 450.16,Z 709.951,A -85,B 0,C 180,E1 9727.428,E2 9727.428} C_VEL
LIN {X 0,Y 455.037,Z 683.323,A -85,B 0,C 180,E1 9727.005,E2 9727.005} C_VEL
LIN {X 0,Y 453.337,Z 685.684,A -85,B 0,C 180,E1 9724.943,E2 9724.943} C_VEL
LIN {X 0,Y 445.496,Z 722.422,A -85,B 0,C 180,E1 9722.38,E2 9722.38} C_VEL
LIN {X 0,Y 439.04,Z 753.45,A -85,B 0,C 180,E1 9720.033,E2 9720.033} C_VEL
LIN {X 0,Y 433.62,Z 780.993,A -85,B 0,C 180,E1 9717.621,E2 9717.621} C_VEL
LIN {X 0,Y 428.853,Z 808.446,A -85,B 0,C 180,E1 9714.833,E2 9714.833} C_VEL
LIN {X 0,Y 425.53,Z 832.079,A -85,B 0,C 180,E1 9712.082,E2 9712.082} C_VEL
LIN {X 0,Y 424.219,Z 842.816,A -85,B 0,C 180,E1 9710.756,E2 9710.756} C_VEL
